METHOD PUBLIC Clone : I_Node
VAR
	pNode : POINTER TO NE_LWORD;
END_VAR
pNode := __NEW(NE_LWORD);
Clone := pNode^;
END_METHOD

METHOD FB_init : BOOL
VAR_INPUT
	bInitRetains : BOOL; // if TRUE, the retain variables are initialized (warm start / cold start)
	bInCopyCode : BOOL;  // if TRUE, the instance afterwards gets moved into the copy code (online change)
END_VAR
AddInput('in1',THIS^.in1);
AddInput('in2',THIS^.in2);
AddOutput('out', THIS^.out);
END_METHOD

METHOD PROTECTED OnExecute
VAR
END_VAR
out.Value := in1.Value <> in2.Value;
END_METHOD

END_FUNCTION_BLOCK

// ---- Comparison/Nodes/NE/NE_REAL.TcPOU
{attribute 'linkalways'} 
{attribute 'no_explicit_call' := 'This FB is a CLASS and must be accessed using methods or properties'}
{attribute 'enable_dynamic_creation'}
FUNCTION_BLOCK FINAL NE_REAL EXTENDS Node
VAR
	in1 : _REAL(0.0);
	in2 : _REAL(0.0);
	out : _BOOL(FALSE);
END_VAR

METHOD PUBLIC Clone : I_Node
VAR
	pNode : POINTER TO NE_REAL;
END_VAR
pNode := __NEW(NE_REAL);
Clone := pNode^;
END_METHOD

METHOD FB_init : BOOL
VAR_INPUT
	bInitRetains : BOOL; // if TRUE, the retain variables are initialized (warm start / cold start)
	bInCopyCode : BOOL;  // if TRUE, the instance afterwards gets moved into the copy code (online change)
END_VAR
AddInput('in1',THIS^.in1);
AddInput('in2',THIS^.in2);
AddOutput('out', THIS^.out);
END_METHOD

METHOD PROTECTED OnExecute
VAR
END_VAR
out.Value := in1.Value <> in2.Value;
END_METHOD

END_FUNCTION_BLOCK

// ---- Comparison/Nodes/NE/NE_SINT.TcPOU
{attribute 'linkalways'} 
{attribute 'no_explicit_call' := 'This FB is a CLASS and must be accessed using methods or properties'}
{attribute 'enable_dynamic_creation'}
FUNCTION_BLOCK FINAL NE_SINT EXTENDS Node
VAR
	in1 : _SINT(0);
	in2 : _SINT(0);
	out : _BOOL(FALSE);
END_VAR

METHOD PUBLIC Clone : I_Node
VAR
	pNode : POINTER TO NE_SINT;
END_VAR
pNode := __NEW(NE_SINT);
Clone := pNode^;
END_METHOD

METHOD FB_init : BOOL
VAR_INPUT
	bInitRetains : BOOL; // if TRUE, the retain variables are initialized (warm start / cold start)
	bInCopyCode : BOOL;  // if TRUE, the instance afterwards gets moved into the copy code (online change)
END_VAR
AddInput('in1',THIS^.in1);
AddInput('in2',THIS^.in2);
AddOutput('out', THIS^.out);
END_METHOD

METHOD PROTECTED OnExecute
VAR
END_VAR
out.Value := in1.Value <> in2.Value;
END_METHOD

END_FUNCTION_BLOCK

// ---- Comparison/Nodes/NE/NE_UDINT.TcPOU
{attribute 'linkalways'} 
{attribute 'no_explicit_call' := 'This FB is a CLASS and must be accessed using methods or properties'}
{attribute 'enable_dynamic_creation'}
FUNCTION_BLOCK FINAL NE_UDINT EXTENDS Node
VAR
	in1 : _UDINT(0);
	in2 : _UDINT(0);
	out : _BOOL(FALSE);
END_VAR

METHOD PUBLIC Clone : I_Node
VAR
	pNode : POINTER TO NE_UDINT;
END_VAR
pNode := __NEW(NE_UDINT);
Clone := pNode^;
END_METHOD

METHOD FB_init : BOOL
VAR_INPUT
	bInitRetains : BOOL; // if TRUE, the retain variables are initialized (warm start / cold start)
	bInCopyCode : BOOL;  // if TRUE, the instance afterwards gets moved into the copy code (online change)
END_VAR
AddInput('in1',THIS^.in1);
AddInput('in2',THIS^.in2);
AddOutput('out', THIS^.out);
END_METHOD

METHOD PROTECTED OnExecute
VAR
END_VAR
out.Value := in1.Value <> in2.Value;
END_METHOD

END_FUNCTION_BLOCK

// ---- Comparison/Nodes/NE/NE_UINT.TcPOU
{attribute 'linkalways'} 
{attribute 'no_explicit_call' := 'This FB is a CLASS and must be accessed using methods or properties'}
{attribute 'enable_dynamic_creation'}
FUNCTION_BLOCK FINAL NE_UINT EXTENDS Node
VAR
	in1 : _UINT(0);
	in2 : _UINT(0);
	out : _BOOL(FALSE);
END_VAR

METHOD PUBLIC Clone : I_Node
VAR
	pNode : POINTER TO NE_UINT;
END_VAR
pNode := __NEW(NE_UINT);
Clone := pNode^;
END_METHOD

METHOD FB_init : BOOL
VAR_INPUT
	bInitRetains : BOOL; // if TRUE, the retain variables are initialized (warm start / cold start)
	bInCopyCode : BOOL;  // if TRUE, the instance afterwards gets moved into the copy code (online change)
END_VAR
AddInput('in1',THIS^.in1);
AddInput('in2',THIS^.in2);
AddOutput('out', THIS^.out);
END_METHOD

METHOD PROTECTED OnExecute
VAR
END_VAR
out.Value := in1.Value <> in2.Value;
END_METHOD

END_FUNCTION_BLOCK

// ---- Comparison/Nodes/NE/NE_ULINT.TcPOU
{attribute 'linkalways'} 
{attribute 'no_explicit_call' := 'This FB is a CLASS and must be accessed using methods or properties'}
{attribute 'enable_dynamic_creation'}
FUNCTION_BLOCK FINAL NE_ULINT EXTENDS Node
VAR
	in1 : _ULINT(0);
	in2 : _ULINT(0);
	out : _BOOL(FALSE);
END_VAR

METHOD PUBLIC Clone : I_Node
VAR
	pNode : POINTER TO NE_ULINT;
END_VAR
pNode := __NEW(NE_ULINT);
Clone := pNode^;
END_METHOD

METHOD FB_init : BOOL
VAR_INPUT
	bInitRetains : BOOL; // if TRUE, the retain variables are initialized (warm start / cold start)
	bInCopyCode : BOOL;  // if TRUE, the instance afterwards gets moved into the copy code (online change)
END_VAR
AddInput('in1',THIS^.in1);
AddInput('in2',THIS^.in2);
AddOutput('out', THIS^.out);
END_METHOD

METHOD PROTECTED OnExecute
VAR
END_VAR
out.Value := in1.Value <> in2.Value;
END_METHOD

END_FUNCTION_BLOCK

// ---- Comparison/Nodes/NE/NE_USINT.TcPOU
{attribute 'linkalways'} 
{attribute 'no_explicit_call' := 'This FB is a CLASS and must be accessed using methods or properties'}
{attribute 'enable_dynamic_creation'}
FUNCTION_BLOCK FINAL NE_USINT EXTENDS Node
VAR
	in1 : _USINT(0);
	in2 : _USINT(0);
	out : _BOOL(FALSE);
END_VAR

METHOD PUBLIC Clone : I_Node
VAR
	pNode : POINTER TO NE_USINT;
END_VAR
pNode := __NEW(NE_USINT);
Clone := pNode^;
END_METHOD

METHOD FB_init : BOOL
VAR_INPUT
	bInitRetains : BOOL; // if TRUE, the retain variables are initialized (warm start / cold start)
	bInCopyCode : BOOL;  // if TRUE, the instance afterwards gets moved into the copy code (online change)
END_VAR
AddInput('in1',THIS^.in1);
AddInput('in2',THIS^.in2);
AddOutput('out', THIS^.out);
END_METHOD

METHOD PROTECTED OnExecute
VAR
END_VAR
out.Value := in1.Value <> in2.Value;
END_METHOD

END_FUNCTION_BLOCK

// ---- Comparison/Nodes/NE/NE_WORD.TcPOU
{attribute 'linkalways'} 
{attribute 'no_explicit_call' := 'This FB is a CLASS and must be accessed using methods or properties'}
{attribute 'enable_dynamic_creation'}
FUNCTION_BLOCK FINAL NE_WORD EXTENDS Node
VAR
	in1 : _WORD(0);
	in2 : _WORD(0);
	out : _BOOL(FALSE);
END_VAR

METHOD PUBLIC Clone : I_Node
VAR
	pNode : POINTER TO NE_WORD;
END_VAR
pNode := __NEW(NE_WORD);
Clone := pNode^;
END_METHOD

METHOD FB_init : BOOL
VAR_INPUT
	bInitRetains : BOOL; // if TRUE, the retain variables are initialized (warm start / cold start)
	bInCopyCode : BOOL;  // if TRUE, the instance afterwards gets moved into the copy code (online change)
END_VAR
AddInput('in1',THIS^.in1);
AddInput('in2',THIS^.in2);
AddOutput('out', THIS^.out);
END_METHOD

METHOD PROTECTED OnExecute
VAR
END_VAR
out.Value := in1.Value <> in2.Value;
END_METHOD

END_FUNCTION_BLOCK

// ---- Core/MathCorePack.TcPOU
{attribute 'linkalways'} 
{attribute 'no_explicit_call' := 'This FB is a CLASS and must be accessed using methods or properties'}
{attribute 'enable_dynamic_creation'}
FUNCTION_BLOCK MathCorePack IMPLEMENTS I_GraphPack
VAR
	ADD_BYTE : ADD_BYTE;
	ADD_DINT : ADD_DINT;
	ADD_DWORD : ADD_DWORD;
	ADD_INT : ADD_INT;
	ADD_LINT : ADD_LINT;
	ADD_LREAL : ADD_LREAL;
	ADD_LWORD : ADD_LWORD;
	ADD_REAL : ADD_REAL;
	ADD_SINT : ADD_SINT;
	ADD_UDINT : ADD_UDINT;
	ADD_UINT : ADD_UINT;
	ADD_ULINT : ADD_ULINT;
	ADD_USINT : ADD_USINT;
	ADD_WORD : ADD_WORD;
	
	SUB_BYTE : SUB_BYTE;
	SUB_DINT : SUB_DINT;
	SUB_DWORD : SUB_DWORD;
	SUB_INT : SUB_INT;
	SUB_LINT : SUB_LINT;
	SUB_LREAL : SUB_LREAL;
	SUB_LWORD : SUB_LWORD;
	SUB_REAL : SUB_REAL;
	SUB_SINT : SUB_SINT;
	SUB_UDINT : SUB_UDINT;
	SUB_UINT : SUB_UINT;
	SUB_ULINT : SUB_ULINT;
	SUB_USINT : SUB_USINT;
	SUB_WORD : SUB_WORD;
	
	MUL_BYTE : MUL_BYTE;
	MUL_DINT : MUL_DINT;
	MUL_DWORD : MUL_DWORD;
	MUL_INT : MUL_INT;
	MUL_LINT : MUL_LINT;
	MUL_LREAL : MUL_LREAL;
	MUL_LWORD : MUL_LWORD;
	MUL_REAL : MUL_REAL;
	MUL_SINT : MUL_SINT;
	MUL_UDINT : MUL_UDINT;
	MUL_UINT : MUL_UINT;
	MUL_ULINT : MUL_ULINT;
	MUL_USINT : MUL_USINT;
	MUL_WORD : MUL_WORD;
	
	DIV_BYTE : DIV_BYTE;
	DIV_DINT : DIV_DINT;
	DIV_DWORD : DIV_DWORD;
	DIV_INT : DIV_INT;
	DIV_LINT : DIV_LINT;
	DIV_LREAL : DIV_LREAL;
	DIV_LWORD : DIV_LWORD;
	DIV_REAL : DIV_REAL;
	DIV_SINT : DIV_SINT;
	DIV_UDINT : DIV_UDINT;
	DIV_UINT : DIV_UINT;
	DIV_ULINT : DIV_ULINT;
	DIV_USINT : DIV_USINT;
	DIV_WORD : DIV_WORD;
	
	MOD_BYTE : MOD_BYTE;
	MOD_DINT : MOD_DINT;
	MOD_DWORD : MOD_DWORD;
	MOD_INT : MOD_INT;
	MOD_LINT : MOD_LINT;
	MOD_LREAL : MOD_LREAL;
	MOD_LWORD : MOD_LWORD;
	MOD_SINT : MOD_SINT;
	MOD_UDINT : MOD_UDINT;
	MOD_UINT : MOD_UINT;
	MOD_ULINT : MOD_ULINT;
	MOD_USINT : MOD_USINT;
	MOD_WORD : MOD_WORD;
	

END_VAR

METHOD Register
VAR_INPUT
	Datatypes : I_Datatypes;
	NodeFactory : I_NodeFactory;
END_VAR
NodeFactory.AddNodeAsPrototype('Math/Core/ADD/ADD_BYTE',ADD_BYTE);
NodeFactory.AddNodeAsPrototype('Math/Core/ADD/ADD_DINT',ADD_DINT);
NodeFactory.AddNodeAsPrototype('Math/Core/ADD/ADD_DWORD',ADD_DWORD);
NodeFactory.AddNodeAsPrototype('Math/Core/ADD/ADD_INT',ADD_INT);
NodeFactory.AddNodeAsPrototype('Math/Core/ADD/ADD_LINT',ADD_LINT);
NodeFactory.AddNodeAsPrototype('Math/Core/ADD/ADD_LREAL',ADD_LREAL);
NodeFactory.AddNodeAsPrototype('Math/Core/ADD/ADD_LWORD',ADD_LWORD);
NodeFactory.AddNodeAsPrototype('Math/Core/ADD/ADD_REAL',ADD_REAL);
NodeFactory.AddNodeAsPrototype('Math/Core/ADD/ADD_SINT',ADD_SINT);
NodeFactory.AddNodeAsPrototype('Math/Core/ADD/ADD_UDINT',ADD_UDINT);
NodeFactory.AddNodeAsPrototype('Math/Core/ADD/ADD_UINT',ADD_UINT);
NodeFactory.AddNodeAsPrototype('Math/Core/ADD/ADD_ULINT',ADD_ULINT);
NodeFactory.AddNodeAsPrototype('Math/Core/ADD/ADD_USINT',ADD_USINT);
NodeFactory.AddNodeAsPrototype('Math/Core/ADD/ADD_WORD',ADD_WORD);

NodeFactory.AddNodeAsPrototype('Math/Core/SUB/SUB_BYTE',SUB_BYTE);
NodeFactory.AddNodeAsPrototype('Math/Core/SUB/SUB_DINT',SUB_DINT);
NodeFactory.AddNodeAsPrototype('Math/Core/SUB/SUB_DWORD',SUB_DWORD);
NodeFactory.AddNodeAsPrototype('Math/Core/SUB/SUB_INT',SUB_INT);
NodeFactory.AddNodeAsPrototype('Math/Core/SUB/SUB_LINT',SUB_LINT);
NodeFactory.AddNodeAsPrototype('Math/Core/SUB/SUB_LREAL',SUB_LREAL);
NodeFactory.AddNodeAsPrototype('Math/Core/SUB/SUB_LWORD',SUB_LWORD);
NodeFactory.AddNodeAsPrototype('Math/Core/SUB/SUB_REAL',SUB_REAL);
NodeFactory.AddNodeAsPrototype('Math/Core/SUB/SUB_SINT',SUB_SINT);
NodeFactory.AddNodeAsPrototype('Math/Core/SUB/SUB_UDINT',SUB_UDINT);
NodeFactory.AddNodeAsPrototype('Math/Core/SUB/SUB_UINT',SUB_UINT);
NodeFactory.AddNodeAsPrototype('Math/Core/SUB/SUB_ULINT',SUB_ULINT);
NodeFactory.AddNodeAsPrototype('Math/Core/SUB/SUB_USINT',SUB_USINT);
NodeFactory.AddNodeAsPrototype('Math/Core/SUB/SUB_WORD',SUB_WORD);

NodeFactory.AddNodeAsPrototype('Math/Core/MUL/MUL_BYTE',MUL_BYTE);
NodeFactory.AddNodeAsPrototype('Math/Core/MUL/MUL_DINT',MUL_DINT);
NodeFactory.AddNodeAsPrototype('Math/Core/MUL/MUL_DWORD',MUL_DWORD);
NodeFactory.AddNodeAsPrototype('Math/Core/MUL/MUL_INT',MUL_INT);
NodeFactory.AddNodeAsPrototype('Math/Core/MUL/MUL_LINT',MUL_LINT);
NodeFactory.AddNodeAsPrototype('Math/Core/MUL/MUL_LREAL',MUL_LREAL);
NodeFactory.AddNodeAsPrototype('Math/Core/MUL/MUL_LWORD',MUL_LWORD);
NodeFactory.AddNodeAsPrototype('Math/Core/MUL/MUL_REAL',MUL_REAL);
NodeFactory.AddNodeAsPrototype('Math/Core/MUL/MUL_SINT',MUL_SINT);
NodeFactory.AddNodeAsPrototype('Math/Core/MUL/MUL_UDINT',MUL_UDINT);
NodeFactory.AddNodeAsPrototype('Math/Core/MUL/MUL_UINT',MUL_UINT);
NodeFactory.AddNodeAsPrototype('Math/Core/MUL/MUL_ULINT',MUL_ULINT);
NodeFactory.AddNodeAsPrototype('Math/Core/MUL/MUL_USINT',MUL_USINT);
NodeFactory.AddNodeAsPrototype('Math/Core/MUL/MUL_WORD',MUL_WORD);

NodeFactory.AddNodeAsPrototype('Math/Core/DIV/DIV_BYTE',DIV_BYTE);
NodeFactory.AddNodeAsPrototype('Math/Core/DIV/DIV_DINT',DIV_DINT);
NodeFactory.AddNodeAsPrototype('Math/Core/DIV/DIV_DWORD',DIV_DWORD);
NodeFactory.AddNodeAsPrototype('Math/Core/DIV/DIV_INT',DIV_INT);
NodeFactory.AddNodeAsPrototype('Math/Core/DIV/DIV_LINT',DIV_LINT);
NodeFactory.AddNodeAsPrototype('Math/Core/DIV/DIV_LREAL',DIV_LREAL);
NodeFactory.AddNodeAsPrototype('Math/Core/DIV/DIV_LWORD',DIV_LWORD);
NodeFactory.AddNodeAsPrototype('Math/Core/DIV/DIV_REAL',DIV_REAL);
NodeFactory.AddNodeAsPrototype('Math/Core/DIV/DIV_SINT',DIV_SINT);
NodeFactory.AddNodeAsPrototype('Math/Core/DIV/DIV_UDINT',DIV_UDINT);
NodeFactory.AddNodeAsPrototype('Math/Core/DIV/DIV_UINT',DIV_UINT);
NodeFactory.AddNodeAsPrototype('Math/Core/DIV/DIV_ULINT',DIV_ULINT);
NodeFactory.AddNodeAsPrototype('Math/Core/DIV/DIV_USINT',DIV_USINT);
NodeFactory.AddNodeAsPrototype('Math/Core/DIV/DIV_WORD',DIV_WORD);

NodeFactory.AddNodeAsPrototype('Math/Core/MOD/MOD_BYTE',MOD_BYTE);
NodeFactory.AddNodeAsPrototype('Math/Core/MOD/MOD_DINT',MOD_DINT);
NodeFactory.AddNodeAsPrototype('Math/Core/MOD/MOD_DWORD',MOD_DWORD);
NodeFactory.AddNodeAsPrototype('Math/Core/MOD/MOD_INT',MOD_INT);
NodeFactory.AddNodeAsPrototype('Math/Core/MOD/MOD_LINT',MOD_LINT);
NodeFactory.AddNodeAsPrototype('Math/Core/MOD/MOD_LREAL',MOD_LREAL);
NodeFactory.AddNodeAsPrototype('Math/Core/MOD/MOD_LWORD',MOD_LWORD);
NodeFactory.AddNodeAsPrototype('Math/Core/MOD/MOD_SINT',MOD_SINT);
NodeFactory.AddNodeAsPrototype('Math/Core/MOD/MOD_UDINT',MOD_UDINT);
NodeFactory.AddNodeAsPrototype('Math/Core/MOD/MOD_UINT',MOD_UINT);
NodeFactory.AddNodeAsPrototype('Math/Core/MOD/MOD_ULINT',MOD_ULINT);
NodeFactory.AddNodeAsPrototype('Math/Core/MOD/MOD_USINT',MOD_USINT);
NodeFactory.AddNodeAsPrototype('Math/Core/MOD/MOD_WORD',MOD_WORD);
END_METHOD

END_FUNCTION_BLOCK

// ---- Core/Nodes/ADD/ADD_BYTE.TcPOU
{attribute 'linkalways'} 
{attribute 'no_explicit_call' := 'This FB is a CLASS and must be accessed using methods or properties'}
{attribute 'enable_dynamic_creation'}
FUNCTION_BLOCK FINAL ADD_BYTE EXTENDS Node
VAR
	in1 : _BYTE(0);
	in2 : _BYTE(0);
	out : _BYTE(0);
END_VAR

METHOD PUBLIC Clone : I_Node
VAR
	pNode : POINTER TO ADD_BYTE;
END_VAR
pNode := __NEW(ADD_BYTE);
Clone := pNode^;
END_METHOD

METHOD FB_init : BOOL
VAR_INPUT
	bInitRetains : BOOL; // if TRUE, the retain variables are initialized (warm start / cold start)
	bInCopyCode : BOOL;  // if TRUE, the instance afterwards gets moved into the copy code (online change)
END_VAR
AddInput('in1',THIS^.in1);
AddInput('in2',THIS^.in2);
AddOutput('out', THIS^.out);
END_METHOD

METHOD PROTECTED OnExecute
VAR
END_VAR
out.Value := in1.Value + in2.Value;
END_METHOD

END_FUNCTION_BLOCK

// ---- Core/Nodes/ADD/ADD_DINT.TcPOU
{attribute 'linkalways'} 
{attribute 'no_explicit_call' := 'This FB is a CLASS and must be accessed using methods or properties'}
{attribute 'enable_dynamic_creation'}
FUNCTION_BLOCK FINAL ADD_DINT EXTENDS Node
VAR
	in1 : _DINT(0);
	in2 : _DINT(0);
	out : _DINT(0);
END_VAR

METHOD PUBLIC Clone : I_Node
VAR
	pNode : POINTER TO ADD_DINT;
END_VAR
pNode := __NEW(ADD_DINT);
Clone := pNode^;
END_METHOD

METHOD FB_init : BOOL
VAR_INPUT
	bInitRetains : BOOL; // if TRUE, the retain variables are initialized (warm start / cold start)
	bInCopyCode : BOOL;  // if TRUE, the instance afterwards gets moved into the copy code (online change)
END_VAR
AddInput('in1',THIS^.in1);
AddInput('in2',THIS^.in2);
AddOutput('out', THIS^.out);
END_METHOD

METHOD PROTECTED OnExecute
VAR
END_VAR
out.Value := in1.Value + in2.Value;
END_METHOD

END_FUNCTION_BLOCK

// ---- Core/Nodes/ADD/ADD_DWORD.TcPOU
{attribute 'linkalways'} 
{attribute 'no_explicit_call' := 'This FB is a CLASS and must be accessed using methods or properties'}
{attribute 'enable_dynamic_creation'}
FUNCTION_BLOCK FINAL ADD_DWORD EXTENDS Node
VAR
	in1 : _DWORD(0);
	in2 : _DWORD(0);
	out : _DWORD(0);
END_VAR

METHOD PUBLIC Clone : I_Node
VAR
	pNode : POINTER TO ADD_DWORD;
END_VAR
pNode := __NEW(ADD_DWORD);
Clone := pNode^;
END_METHOD

METHOD FB_init : BOOL
VAR_INPUT
	bInitRetains : BOOL; // if TRUE, the retain variables are initialized (warm start / cold start)
	bInCopyCode : BOOL;  // if TRUE, the instance afterwards gets moved into the copy code (online change)
END_VAR
AddInput('in1',THIS^.in1);
AddInput('in2',THIS^.in2);
AddOutput('out', THIS^.out);
END_METHOD

METHOD PROTECTED OnExecute
VAR
END_VAR
out.Value := in1.Value + in2.Value;
END_METHOD

END_FUNCTION_BLOCK

// ---- Core/Nodes/ADD/ADD_INT.TcPOU
{attribute 'linkalways'} 
{attribute 'no_explicit_call' := 'This FB is a CLASS and must be accessed using methods or properties'}
{attribute 'enable_dynamic_creation'}
FUNCTION_BLOCK FINAL ADD_INT EXTENDS Node
VAR
	in1 : _INT(0);
	in2 : _INT(0);
	out : _INT(0);
END_VAR

METHOD PUBLIC Clone : I_Node
VAR
	pNode : POINTER TO ADD_INT;
END_VAR
pNode := __NEW(ADD_INT);
Clone := pNode^;
END_METHOD

METHOD FB_init : BOOL
VAR_INPUT
	bInitRetains : BOOL; // if TRUE, the retain variables are initialized (warm start / cold start)
	bInCopyCode : BOOL;  // if TRUE, the instance afterwards gets moved into the copy code (online change)
END_VAR
AddInput('in1',THIS^.in1);
AddInput('in2',THIS^.in2);
AddOutput('out', THIS^.out);
END_METHOD

METHOD PROTECTED OnExecute
VAR
END_VAR
out.Value := in1.Value + in2.Value;
END_METHOD

END_FUNCTION_BLOCK

// ---- Core/Nodes/ADD/ADD_LINT.TcPOU
{attribute 'linkalways'} 
{attribute 'no_explicit_call' := 'This FB is a CLASS and must be accessed using methods or properties'}
{attribute 'enable_dynamic_creation'}
FUNCTION_BLOCK FINAL ADD_LINT EXTENDS Node
VAR
	in1 : _LINT(0);
	in2 : _LINT(0);
	out : _LINT(0);
END_VAR

METHOD PUBLIC Clone : I_Node
VAR
	pNode : POINTER TO ADD_LINT;
END_VAR
pNode := __NEW(ADD_LINT);
Clone := pNode^;
END_METHOD

METHOD FB_init : BOOL
VAR_INPUT
	bInitRetains : BOOL; // if TRUE, the retain variables are initialized (warm start / cold start)
	bInCopyCode : BOOL;  // if TRUE, the instance afterwards gets moved into the copy code (online change)
END_VAR
AddInput('in1',THIS^.in1);
AddInput('in2',THIS^.in2);
AddOutput('out', THIS^.out);
END_METHOD

METHOD PROTECTED OnExecute
VAR
END_VAR
out.Value := in1.Value + in2.Value;
END_METHOD

END_FUNCTION_BLOCK

// ---- Core/Nodes/ADD/ADD_LREAL.TcPOU
{attribute 'linkalways'} 
{attribute 'no_explicit_call' := 'This FB is a CLASS and must be accessed using methods or properties'}
{attribute 'enable_dynamic_creation'}
FUNCTION_BLOCK FINAL ADD_LREAL EXTENDS Node
VAR
	in1 : _LREAL(0.0);
	in2 : _LREAL(0.0);
	out : _LREAL(0.0);
END_VAR

METHOD PUBLIC Clone : I_Node
VAR
	pNode : POINTER TO ADD_LREAL;
END_VAR
pNode := __NEW(ADD_LREAL);
Clone := pNode^;
END_METHOD

METHOD FB_init : BOOL
VAR_INPUT
	bInitRetains : BOOL; // if TRUE, the retain variables are initialized (warm start / cold start)
	bInCopyCode : BOOL;  // if TRUE, the instance afterwards gets moved into the copy code (online change)
END_VAR
AddInput('in1',THIS^.in1);
AddInput('in2',THIS^.in2);
AddOutput('out', THIS^.out);
END_METHOD

METHOD PROTECTED OnExecute
VAR
END_VAR
out.Value := in1.Value + in2.Value;
END_METHOD

END_FUNCTION_BLOCK

// ---- Core/Nodes/ADD/ADD_LWORD.TcPOU
{attribute 'linkalways'} 
{attribute 'no_explicit_call' := 'This FB is a CLASS and must be accessed using methods or properties'}
{attribute 'enable_dynamic_creation'}
FUNCTION_BLOCK FINAL ADD_LWORD EXTENDS Node
VAR
	in1 : _LWORD(0);
	in2 : _LWORD(0);
	out : _LWORD(0);
END_VAR

METHOD PUBLIC Clone : I_Node
VAR
	pNode : POINTER TO ADD_LWORD;
END_VAR
pNode := __NEW(ADD_LWORD);
Clone := pNode^;
END_METHOD

METHOD FB_init : BOOL
VAR_INPUT
	bInitRetains : BOOL; // if TRUE, the retain variables are initialized (warm start / cold start)
	bInCopyCode : BOOL;  // if TRUE, the instance afterwards gets moved into the copy code (online change)
END_VAR
AddInput('in1',THIS^.in1);
AddInput('in2',THIS^.in2);
AddOutput('out', THIS^.out);
END_METHOD

METHOD PROTECTED OnExecute
VAR
END_VAR
out.Value := in1.Value + in2.Value;
END_METHOD

END_FUNCTION_BLOCK

// ---- Core/Nodes/ADD/ADD_REAL.TcPOU
{attribute 'linkalways'} 
{attribute 'no_explicit_call' := 'This FB is a CLASS and must be accessed using methods or properties'}
{attribute 'enable_dynamic_creation'}
FUNCTION_BLOCK FINAL ADD_REAL EXTENDS Node
VAR
	in1 : _REAL(0.0);
	in2 : _REAL(0.0);
	out : _REAL(0.0);
END_VAR

METHOD PUBLIC Clone : I_Node
VAR
	pNode : POINTER TO ADD_REAL;
END_VAR
pNode := __NEW(ADD_REAL);
Clone := pNode^;
END_METHOD

METHOD FB_init : BOOL
VAR_INPUT
	bInitRetains : BOOL; // if TRUE, the retain variables are initialized (warm start / cold start)
	bInCopyCode : BOOL;  // if TRUE, the instance afterwards gets moved into the copy code (online change)
END_VAR
AddInput('in1',THIS^.in1);
AddInput('in2',THIS^.in2);
AddOutput('out', THIS^.out);
END_METHOD

METHOD PROTECTED OnExecute
VAR
END_VAR
out.Value := in1.Value + in2.Value;
END_METHOD

END_FUNCTION_BLOCK

// ---- Core/Nodes/ADD/ADD_SINT.TcPOU
{attribute 'linkalways'} 
{attribute 'no_explicit_call' := 'This FB is a CLASS and must be accessed using methods or properties'}
{attribute 'enable_dynamic_creation'}
FUNCTION_BLOCK FINAL ADD_SINT EXTENDS Node
VAR
	in1 : _SINT(0);
	in2 : _SINT(0);
	out : _SINT(0);
END_VAR

METHOD PUBLIC Clone : I_Node
VAR
	pNode : POINTER TO ADD_SINT;
END_VAR
pNode := __NEW(ADD_SINT);
Clone := pNode^;
END_METHOD

METHOD FB_init : BOOL
VAR_INPUT
	bInitRetains : BOOL; // if TRUE, the retain variables are initialized (warm start / cold start)
	bInCopyCode : BOOL;  // if TRUE, the instance afterwards gets moved into the copy code (online change)
END_VAR
AddInput('in1',THIS^.in1);
AddInput('in2',THIS^.in2);
AddOutput('out', THIS^.out);
END_METHOD

METHOD PROTECTED OnExecute
VAR
END_VAR
out.Value := in1.Value + in2.Value;
END_METHOD

END_FUNCTION_BLOCK

// ---- Core/Nodes/ADD/ADD_UDINT.TcPOU
{attribute 'linkalways'} 
{attribute 'no_explicit_call' := 'This FB is a CLASS and must be accessed using methods or properties'}
{attribute 'enable_dynamic_creation'}
FUNCTION_BLOCK FINAL ADD_UDINT EXTENDS Node
VAR
	in1 : _UDINT(0);
	in2 : _UDINT(0);
	out : _UDINT(0);
END_VAR

METHOD PUBLIC Clone : I_Node
VAR
	pNode : POINTER TO ADD_UDINT;
END_VAR
pNode := __NEW(ADD_UDINT);
Clone := pNode^;
END_METHOD

METHOD FB_init : BOOL
VAR_INPUT
	bInitRetains : BOOL; // if TRUE, the retain variables are initialized (warm start / cold start)
	bInCopyCode : BOOL;  // if TRUE, the instance afterwards gets moved into the copy code (online change)
END_VAR
AddInput('in1',THIS^.in1);
AddInput('in2',THIS^.in2);
AddOutput('out', THIS^.out);
END_METHOD

METHOD PROTECTED OnExecute
VAR
END_VAR
out.Value := in1.Value + in2.Value;
END_METHOD

END_FUNCTION_BLOCK

// ---- Core/Nodes/ADD/ADD_UINT.TcPOU
{attribute 'linkalways'} 
{attribute 'no_explicit_call' := 'This FB is a CLASS and must be accessed using methods or properties'}
{attribute 'enable_dynamic_creation'}
FUNCTION_BLOCK FINAL ADD_UINT EXTENDS Node
VAR
	in1 : _UINT(0);
	in2 : _UINT(0);
	out : _UINT(0);
END_VAR

METHOD PUBLIC Clone : I_Node
VAR
	pNode : POINTER TO ADD_UINT;
END_VAR
pNode := __NEW(ADD_UINT);
Clone := pNode^;
END_METHOD

METHOD FB_init : BOOL
VAR_INPUT
	bInitRetains : BOOL; // if TRUE, the retain variables are initialized (warm start / cold start)
	bInCopyCode : BOOL;  // if TRUE, the instance afterwards gets moved into the copy code (online change)
END_VAR
AddInput('in1',THIS^.in1);
AddInput('in2',THIS^.in2);
AddOutput('out', THIS^.out);
END_METHOD

METHOD PROTECTED OnExecute
VAR
END_VAR
out.Value := in1.Value + in2.Value;
END_METHOD

END_FUNCTION_BLOCK

// ---- Core/Nodes/ADD/ADD_ULINT.TcPOU
{attribute 'linkalways'} 
{attribute 'no_explicit_call' := 'This FB is a CLASS and must be accessed using methods or properties'}
{attribute 'enable_dynamic_creation'}
FUNCTION_BLOCK FINAL ADD_ULINT EXTENDS Node
VAR
	in1 : _ULINT(0);
	in2 : _ULINT(0);
	out : _ULINT(0);
END_VAR

METHOD PUBLIC Clone : I_Node
VAR
	pNode : POINTER TO ADD_ULINT;
END_VAR
pNode := __NEW(ADD_ULINT);
Clone := pNode^;
END_METHOD

METHOD FB_init : BOOL
VAR_INPUT
	bInitRetains : BOOL; // if TRUE, the retain variables are initialized (warm start / cold start)
	bInCopyCode : BOOL;  // if TRUE, the instance afterwards gets moved into the copy code (online change)
END_VAR
AddInput('in1',THIS^.in1);
AddInput('in2',THIS^.in2);
AddOutput('out', THIS^.out);
END_METHOD

METHOD PROTECTED OnExecute
VAR
END_VAR
out.Value := in1.Value + in2.Value;
END_METHOD

END_FUNCTION_BLOCK

// ---- Core/Nodes/ADD/ADD_USINT.TcPOU
{attribute 'linkalways'} 
{attribute 'no_explicit_call' := 'This FB is a CLASS and must be accessed using methods or properties'}
{attribute 'enable_dynamic_creation'}
FUNCTION_BLOCK FINAL ADD_USINT EXTENDS Node
VAR
	in1 : _USINT(0);
	in2 : _USINT(0);
	out : _USINT(0);
END_VAR

METHOD PUBLIC Clone : I_Node
VAR
	pNode : POINTER TO ADD_USINT;
END_VAR
pNode := __NEW(ADD_USINT);
Clone := pNode^;
END_METHOD

METHOD FB_init : BOOL
VAR_INPUT
	bInitRetains : BOOL; // if TRUE, the retain variables are initialized (warm start / cold start)
	bInCopyCode : BOOL;  // if TRUE, the instance afterwards gets moved into the copy code (online change)
END_VAR
AddInput('in1',THIS^.in1);
AddInput('in2',THIS^.in2);
AddOutput('out', THIS^.out);
END_METHOD

METHOD PROTECTED OnExecute
VAR
END_VAR
out.Value := in1.Value + in2.Value;
END_METHOD

END_FUNCTION_BLOCK

// ---- Core/Nodes/ADD/ADD_WORD.TcPOU
{attribute 'linkalways'} 
{attribute 'no_explicit_call' := 'This FB is a CLASS and must be accessed using methods or properties'}
{attribute 'enable_dynamic_creation'}
FUNCTION_BLOCK FINAL ADD_WORD EXTENDS Node
VAR
	in1 : _WORD(0);
	in2 : _WORD(0);
	out : _WORD(0);
END_VAR

METHOD PUBLIC Clone : I_Node
VAR
	pNode : POINTER TO ADD_WORD;
END_VAR
pNode := __NEW(ADD_WORD);
Clone := pNode^;
END_METHOD

METHOD FB_init : BOOL
VAR_INPUT
	bInitRetains : BOOL; // if TRUE, the retain variables are initialized (warm start / cold start)
	bInCopyCode : BOOL;  // if TRUE, the instance afterwards gets moved into the copy code (online change)
END_VAR
AddInput('in1',THIS^.in1);
AddInput('in2',THIS^.in2);
AddOutput('out', THIS^.out);
END_METHOD

METHOD PROTECTED OnExecute
VAR
END_VAR
out.Value := in1.Value + in2.Value;
END_METHOD

END_FUNCTION_BLOCK

// ---- Core/Nodes/SUB/SUB_BYTE.TcPOU
{attribute 'linkalways'} 
{attribute 'no_explicit_call' := 'This FB is a CLASS and must be accessed using methods or properties'}
{attribute 'enable_dynamic_creation'}
FUNCTION_BLOCK FINAL SUB_BYTE EXTENDS Node
VAR
	in1 : _BYTE(0);
	in2 : _BYTE(0);
	out : _BYTE(0);
END_VAR

METHOD PUBLIC Clone : I_Node
VAR
	pNode : POINTER TO SUB_BYTE;
END_VAR
pNode := __NEW(SUB_BYTE);
Clone := pNode^;
END_METHOD

METHOD FB_init : BOOL
VAR_INPUT
	bInitRetains : BOOL; // if TRUE, the retain variables are initialized (warm start / cold start)
	bInCopyCode : BOOL;  // if TRUE, the instance afterwards gets moved into the copy code (online change)
END_VAR
AddInput('in1',THIS^.in1);
AddInput('in2',THIS^.in2);
AddOutput('out', THIS^.out);
END_METHOD

METHOD PROTECTED OnExecute
VAR
END_VAR
out.Value := in1.Value - in2.Value;
END_METHOD

END_FUNCTION_BLOCK

// ---- Core/Nodes/SUB/SUB_DINT.TcPOU
{attribute 'linkalways'} 
{attribute 'no_explicit_call' := 'This FB is a CLASS and must be accessed using methods or properties'}
{attribute 'enable_dynamic_creation'}
FUNCTION_BLOCK FINAL SUB_DINT EXTENDS Node
VAR
	in1 : _DINT(0);
	in2 : _DINT(0);
	out : _DINT(0);
END_VAR

METHOD PUBLIC Clone : I_Node
VAR
	pNode : POINTER TO SUB_DINT;
END_VAR
pNode := __NEW(SUB_DINT);
Clone := pNode^;
END_METHOD

METHOD FB_init : BOOL
VAR_INPUT
	bInitRetains : BOOL; // if TRUE, the retain variables are initialized (warm start / cold start)
	bInCopyCode : BOOL;  // if TRUE, the instance afterwards gets moved into the copy code (online change)
END_VAR
AddInput('in1',THIS^.in1);
AddInput('in2',THIS^.in2);
AddOutput('out', THIS^.out);
END_METHOD

METHOD PROTECTED OnExecute
VAR
END_VAR
out.Value := in1.Value - in2.Value;
END_METHOD

END_FUNCTION_BLOCK

// ---- Core/Nodes/SUB/SUB_DWORD.TcPOU
{attribute 'linkalways'} 
{attribute 'no_explicit_call' := 'This FB is a CLASS and must be accessed using methods or properties'}
{attribute 'enable_dynamic_creation'}
FUNCTION_BLOCK FINAL SUB_DWORD EXTENDS Node
VAR
	in1 : _DWORD(0);
	in2 : _DWORD(0);
	out : _DWORD(0);
END_VAR

METHOD PUBLIC Clone : I_Node
VAR
	pNode : POINTER TO SUB_DWORD;
END_VAR
pNode := __NEW(SUB_DWORD);
Clone := pNode^;
END_METHOD

METHOD FB_init : BOOL
VAR_INPUT
	bInitRetains : BOOL; // if TRUE, the retain variables are initialized (warm start / cold start)
	bInCopyCode : BOOL;  // if TRUE, the instance afterwards gets moved into the copy code (online change)
END_VAR
AddInput('in1',THIS^.in1);
AddInput('in2',THIS^.in2);
AddOutput('out', THIS^.out);
END_METHOD

METHOD PROTECTED OnExecute
VAR
END_VAR
out.Value := in1.Value - in2.Value;
END_METHOD

END_FUNCTION_BLOCK

// ---- Core/Nodes/SUB/SUB_INT.TcPOU
{attribute 'linkalways'} 
{attribute 'no_explicit_call' := 'This FB is a CLASS and must be accessed using methods or properties'}
{attribute 'enable_dynamic_creation'}
FUNCTION_BLOCK FINAL SUB_INT EXTENDS Node
VAR
	in1 : _INT(0);
	in2 : _INT(0);
	out : _INT(0);
END_VAR

METHOD PUBLIC Clone : I_Node
VAR
	pNode : POINTER TO SUB_INT;
END_VAR
pNode := __NEW(SUB_INT);
Clone := pNode^;
END_METHOD

METHOD FB_init : BOOL
VAR_INPUT
	bInitRetains : BOOL; // if TRUE, the retain variables are initialized (warm start / cold start)
	bInCopyCode : BOOL;  // if TRUE, the instance afterwards gets moved into the copy code (online change)
END_VAR
AddInput('in1',THIS^.in1);
AddInput('in2',THIS^.in2);
AddOutput('out', THIS^.out);
END_METHOD

METHOD PROTECTED OnExecute
VAR
END_VAR
out.Value := in1.Value - in2.Value;
END_METHOD

END_FUNCTION_BLOCK

// ---- Core/Nodes/SUB/SUB_LINT.TcPOU
{attribute 'linkalways'} 
{attribute 'no_explicit_call' := 'This FB is a CLASS and must be accessed using methods or properties'}
{attribute 'enable_dynamic_creation'}
FUNCTION_BLOCK FINAL SUB_LINT EXTENDS Node
VAR
	in1 : _LINT(0);
	in2 : _LINT(0);
	out : _LINT(0);
END_VAR

METHOD PUBLIC Clone : I_Node
VAR
	pNode : POINTER TO SUB_LINT;
END_VAR
pNode := __NEW(SUB_LINT);
Clone := pNode^;
END_METHOD

METHOD FB_init : BOOL
VAR_INPUT
	bInitRetains : BOOL; // if TRUE, the retain variables are initialized (warm start / cold start)
	bInCopyCode : BOOL;  // if TRUE, the instance afterwards gets moved into the copy code (online change)
END_VAR
AddInput('in1',THIS^.in1);
AddInput('in2',THIS^.in2);
AddOutput('out', THIS^.out);
END_METHOD

METHOD PROTECTED OnExecute
VAR
END_VAR
out.Value := in1.Value - in2.Value;
END_METHOD

END_FUNCTION_BLOCK

// ---- Core/Nodes/SUB/SUB_LREAL.TcPOU
{attribute 'linkalways'} 
{attribute 'no_explicit_call' := 'This FB is a CLASS and must be accessed using methods or properties'}
{attribute 'enable_dynamic_creation'}
FUNCTION_BLOCK FINAL SUB_LREAL EXTENDS Node
VAR
	in1 : _LREAL(0.0);
	in2 : _LREAL(0.0);
	out : _LREAL(0.0);
END_VAR

METHOD PUBLIC Clone : I_Node
VAR
	pNode : POINTER TO SUB_LREAL;
END_VAR
pNode := __NEW(SUB_LREAL);
Clone := pNode^;
END_METHOD

METHOD FB_init : BOOL
VAR_INPUT
	bInitRetains : BOOL; // if TRUE, the retain variables are initialized (warm start / cold start)
	bInCopyCode : BOOL;  // if TRUE, the instance afterwards gets moved into the copy code (online change)
END_VAR
AddInput('in1',THIS^.in1);
AddInput('in2',THIS^.in2);
AddOutput('out', THIS^.out);
END_METHOD

METHOD PROTECTED OnExecute
VAR
END_VAR
out.Value := in1.Value - in2.Value;
END_METHOD

END_FUNCTION_BLOCK

// ---- Core/Nodes/SUB/SUB_LWORD.TcPOU
{attribute 'linkalways'} 
{attribute 'no_explicit_call' := 'This FB is a CLASS and must be accessed using methods or properties'}
{attribute 'enable_dynamic_creation'}
FUNCTION_BLOCK FINAL SUB_LWORD EXTENDS Node
VAR
	in1 : _LWORD(0);
	in2 : _LWORD(0);
	out : _LWORD(0);
END_VAR

METHOD PUBLIC Clone : I_Node
VAR
	pNode : POINTER TO SUB_LWORD;
END_VAR
pNode := __NEW(SUB_LWORD);
Clone := pNode^;
END_METHOD

METHOD FB_init : BOOL
VAR_INPUT
	bInitRetains : BOOL; // if TRUE, the retain variables are initialized (warm start / cold start)
	bInCopyCode : BOOL;  // if TRUE, the instance afterwards gets moved into the copy code (online change)
END_VAR
AddInput('in1',THIS^.in1);
AddInput('in2',THIS^.in2);
AddOutput('out', THIS^.out);
END_METHOD

METHOD PROTECTED OnExecute
VAR
END_VAR
out.Value := in1.Value - in2.Value;
END_METHOD

END_FUNCTION_BLOCK

// ---- Core/Nodes/SUB/SUB_REAL.TcPOU
{attribute 'linkalways'} 
{attribute 'no_explicit_call' := 'This FB is a CLASS and must be accessed using methods or properties'}
{attribute 'enable_dynamic_creation'}
FUNCTION_BLOCK FINAL SUB_REAL EXTENDS Node
VAR
	in1 : _REAL(0.0);
	in2 : _REAL(0.0);
	out : _REAL(0.0);
END_VAR

METHOD PUBLIC Clone : I_Node
VAR
	pNode : POINTER TO SUB_REAL;
END_VAR
pNode := __NEW(SUB_REAL);
Clone := pNode^;
END_METHOD

METHOD FB_init : BOOL
VAR_INPUT
	bInitRetains : BOOL; // if TRUE, the retain variables are initialized (warm start / cold start)
	bInCopyCode : BOOL;  // if TRUE, the instance afterwards gets moved into the copy code (online change)
END_VAR
AddInput('in1',THIS^.in1);
AddInput('in2',THIS^.in2);
AddOutput('out', THIS^.out);
END_METHOD

METHOD PROTECTED OnExecute
VAR
END_VAR
out.Value := in1.Value - in2.Value;
END_METHOD

END_FUNCTION_BLOCK

// ---- Core/Nodes/SUB/SUB_SINT.TcPOU
{attribute 'linkalways'} 
{attribute 'no_explicit_call' := 'This FB is a CLASS and must be accessed using methods or properties'}
{attribute 'enable_dynamic_creation'}
FUNCTION_BLOCK FINAL SUB_SINT EXTENDS Node
VAR
	in1 : _SINT(0);
	in2 : _SINT(0);
	out : _SINT(0);
END_VAR

METHOD PUBLIC Clone : I_Node
VAR
	pNode : POINTER TO SUB_SINT;
END_VAR
pNode := __NEW(SUB_SINT);
Clone := pNode^;
END_METHOD

METHOD FB_init : BOOL
VAR_INPUT
	bInitRetains : BOOL; // if TRUE, the retain variables are initialized (warm start / cold start)
	bInCopyCode : BOOL;  // if TRUE, the instance afterwards gets moved into the copy code (online change)
END_VAR
AddInput('in1',THIS^.in1);
AddInput('in2',THIS^.in2);
AddOutput('out', THIS^.out);
END_METHOD

METHOD PROTECTED OnExecute
VAR
END_VAR
out.Value := in1.Value - in2.Value;
END_METHOD

END_FUNCTION_BLOCK

// ---- Core/Nodes/SUB/SUB_UDINT.TcPOU
{attribute 'linkalways'} 
{attribute 'no_explicit_call' := 'This FB is a CLASS and must be accessed using methods or properties'}
{attribute 'enable_dynamic_creation'}
FUNCTION_BLOCK FINAL SUB_UDINT EXTENDS Node
VAR
	in1 : _UDINT(0);
	in2 : _UDINT(0);
	out : _UDINT(0);
END_VAR

METHOD PUBLIC Clone : I_Node
VAR
	pNode : POINTER TO SUB_UDINT;
END_VAR
pNode := __NEW(SUB_UDINT);
Clone := pNode^;
END_METHOD

METHOD FB_init : BOOL
VAR_INPUT
	bInitRetains : BOOL; // if TRUE, the retain variables are initialized (warm start / cold start)
	bInCopyCode : BOOL;  // if TRUE, the instance afterwards gets moved into the copy code (online change)
END_VAR
AddInput('in1',THIS^.in1);
AddInput('in2',THIS^.in2);
AddOutput('out', THIS^.out);
END_METHOD

METHOD PROTECTED OnExecute
VAR
END_VAR
out.Value := in1.Value - in2.Value;
END_METHOD

END_FUNCTION_BLOCK

// ---- Core/Nodes/SUB/SUB_UINT.TcPOU
{attribute 'linkalways'} 
{attribute 'no_explicit_call' := 'This FB is a CLASS and must be accessed using methods or properties'}
{attribute 'enable_dynamic_creation'}
FUNCTION_BLOCK FINAL SUB_UINT EXTENDS Node
VAR
	in1 : _UINT(0);
	in2 : _UINT(0);
	out : _UINT(0);
END_VAR

METHOD PUBLIC Clone : I_Node
VAR
	pNode : POINTER TO SUB_UINT;
END_VAR
pNode := __NEW(SUB_UINT);
Clone := pNode^;
END_METHOD

METHOD FB_init : BOOL
VAR_INPUT
	bInitRetains : BOOL; // if TRUE, the retain variables are initialized (warm start / cold start)
	bInCopyCode : BOOL;  // if TRUE, the instance afterwards gets moved into the copy code (online change)
END_VAR
AddInput('in1',THIS^.in1);
AddInput('in2',THIS^.in2);
AddOutput('out', THIS^.out);
END_METHOD

METHOD PROTECTED OnExecute
VAR
END_VAR
out.Value := in1.Value - in2.Value;
END_METHOD

END_FUNCTION_BLOCK

// ---- Core/Nodes/SUB/SUB_ULINT.TcPOU
{attribute 'linkalways'} 
{attribute 'no_explicit_call' := 'This FB is a CLASS and must be accessed using methods or properties'}
{attribute 'enable_dynamic_creation'}
FUNCTION_BLOCK FINAL SUB_ULINT EXTENDS Node
VAR
	in1 : _ULINT(0);
	in2 : _ULINT(0);
	out : _ULINT(0);
END_VAR

METHOD PUBLIC Clone : I_Node
VAR
	pNode : POINTER TO SUB_ULINT;
END_VAR
pNode := __NEW(SUB_ULINT);
Clone := pNode^;
END_METHOD

METHOD FB_init : BOOL
VAR_INPUT
	bInitRetains : BOOL; // if TRUE, the retain variables are initialized (warm start / cold start)
	bInCopyCode : BOOL;  // if TRUE, the instance afterwards gets moved into the copy code (online change)
END_VAR
AddInput('in1',THIS^.in1);
AddInput('in2',THIS^.in2);
AddOutput('out', THIS^.out);
END_METHOD

METHOD PROTECTED OnExecute
VAR
END_VAR
out.Value := in1.Value - in2.Value;
END_METHOD

END_FUNCTION_BLOCK

// ---- Core/Nodes/SUB/SUB_USINT.TcPOU
{attribute 'linkalways'} 
{attribute 'no_explicit_call' := 'This FB is a CLASS and must be accessed using methods or properties'}
{attribute 'enable_dynamic_creation'}
FUNCTION_BLOCK FINAL SUB_USINT EXTENDS Node
VAR
	in1 : _USINT(0);
	in2 : _USINT(0);
	out : _USINT(0);
END_VAR

METHOD PUBLIC Clone : I_Node
VAR
	pNode : POINTER TO SUB_USINT;
END_VAR
pNode := __NEW(SUB_USINT);
Clone := pNode^;
END_METHOD

METHOD FB_init : BOOL
VAR_INPUT
	bInitRetains : BOOL; // if TRUE, the retain variables are initialized (warm start / cold start)
	bInCopyCode : BOOL;  // if TRUE, the instance afterwards gets moved into the copy code (online change)
END_VAR
AddInput('in1',THIS^.in1);
AddInput('in2',THIS^.in2);
AddOutput('out', THIS^.out);
END_METHOD

METHOD PROTECTED OnExecute
VAR
END_VAR
out.Value := in1.Value - in2.Value;
END_METHOD

END_FUNCTION_BLOCK

// ---- Core/Nodes/SUB/SUB_WORD.TcPOU
{attribute 'linkalways'} 
{attribute 'no_explicit_call' := 'This FB is a CLASS and must be accessed using methods or properties'}
{attribute 'enable_dynamic_creation'}
FUNCTION_BLOCK FINAL SUB_WORD EXTENDS Node
VAR
	in1 : _WORD(0);
	in2 : _WORD(0);
	out : _WORD(0);
END_VAR

METHOD PUBLIC Clone : I_Node
VAR
	pNode : POINTER TO SUB_WORD;
END_VAR
pNode := __NEW(SUB_WORD);
Clone := pNode^;
END_METHOD

METHOD FB_init : BOOL
VAR_INPUT
	bInitRetains : BOOL; // if TRUE, the retain variables are initialized (warm start / cold start)
	bInCopyCode : BOOL;  // if TRUE, the instance afterwards gets moved into the copy code (online change)
END_VAR
AddInput('in1',THIS^.in1);
AddInput('in2',THIS^.in2);
AddOutput('out', THIS^.out);
END_METHOD

METHOD PROTECTED OnExecute
VAR
END_VAR
out.Value := in1.Value - in2.Value;
END_METHOD

END_FUNCTION_BLOCK

// ---- Core/Nodes/MUL/MUL_BYTE.TcPOU
{attribute 'linkalways'} 
{attribute 'no_explicit_call' := 'This FB is a CLASS and must be accessed using methods or properties'}
{attribute 'enable_dynamic_creation'}
FUNCTION_BLOCK FINAL MUL_BYTE EXTENDS Node
VAR
	in1 : _BYTE(0);
	in2 : _BYTE(0);
	out : _BYTE(0);
END_VAR

METHOD PUBLIC Clone : I_Node
VAR
	pNode : POINTER TO MUL_BYTE;
END_VAR
pNode := __NEW(MUL_BYTE);
Clone := pNode^;
END_METHOD

METHOD FB_init : BOOL
VAR_INPUT
	bInitRetains : BOOL; // if TRUE, the retain variables are initialized (warm start / cold start)
	bInCopyCode : BOOL;  // if TRUE, the instance afterwards gets moved into the copy code (online change)
END_VAR
AddInput('in1',THIS^.in1);
AddInput('in2',THIS^.in2);
AddOutput('out', THIS^.out);
END_METHOD

METHOD PROTECTED OnExecute
VAR
END_VAR
out.Value := in1.Value * in2.Value;
END_METHOD

END_FUNCTION_BLOCK

// ---- Core/Nodes/MUL/MUL_DINT.TcPOU
{attribute 'linkalways'} 
{attribute 'no_explicit_call' := 'This FB is a CLASS and must be accessed using methods or properties'}
{attribute 'enable_dynamic_creation'}
FUNCTION_BLOCK FINAL MUL_DINT EXTENDS Node
VAR
	in1 : _DINT(0);
	in2 : _DINT(0);
	out : _DINT(0);
END_VAR

METHOD PUBLIC Clone : I_Node
VAR
	pNode : POINTER TO MUL_DINT;
END_VAR
pNode := __NEW(MUL_DINT);
Clone := pNode^;
END_METHOD

METHOD FB_init : BOOL
VAR_INPUT
	bInitRetains : BOOL; // if TRUE, the retain variables are initialized (warm start / cold start)
	bInCopyCode : BOOL;  // if TRUE, the instance afterwards gets moved into the copy code (online change)
END_VAR
AddInput('in1',THIS^.in1);
AddInput('in2',THIS^.in2);
AddOutput('out', THIS^.out);
END_METHOD

METHOD PROTECTED OnExecute
VAR
END_VAR
out.Value := in1.Value * in2.Value;
END_METHOD

END_FUNCTION_BLOCK

// ---- Core/Nodes/MUL/MUL_DWORD.TcPOU
{attribute 'linkalways'} 
{attribute 'no_explicit_call' := 'This FB is a CLASS and must be accessed using methods or properties'}
{attribute 'enable_dynamic_creation'}
FUNCTION_BLOCK FINAL MUL_DWORD EXTENDS Node
VAR
	in1 : _DWORD(0);
	in2 : _DWORD(0);
	out : _DWORD(0);
END_VAR

METHOD PUBLIC Clone : I_Node
VAR
	pNode : POINTER TO MUL_DWORD;
END_VAR
pNode := __NEW(MUL_DWORD);
Clone := pNode^;
END_METHOD

METHOD FB_init : BOOL
VAR_INPUT
	bInitRetains : BOOL; // if TRUE, the retain variables are initialized (warm start / cold start)
	bInCopyCode : BOOL;  // if TRUE, the instance afterwards gets moved into the copy code (online change)
END_VAR
AddInput('in1',THIS^.in1);
AddInput('in2',THIS^.in2);
AddOutput('out', THIS^.out);
END_METHOD

METHOD PROTECTED OnExecute
VAR
END_VAR
out.Value := in1.Value * in2.Value;
END_METHOD

END_FUNCTION_BLOCK

// ---- Core/Nodes/MUL/MUL_INT.TcPOU
{attribute 'linkalways'} 
{attribute 'no_explicit_call' := 'This FB is a CLASS and must be accessed using methods or properties'}
{attribute 'enable_dynamic_creation'}
FUNCTION_BLOCK FINAL MUL_INT EXTENDS Node
VAR
	in1 : _INT(0);
	in2 : _INT(0);
	out : _INT(0);
END_VAR

METHOD PUBLIC Clone : I_Node
VAR
	pNode : POINTER TO MUL_INT;
END_VAR
pNode := __NEW(MUL_INT);
Clone := pNode^;
END_METHOD

METHOD FB_init : BOOL
VAR_INPUT
	bInitRetains : BOOL; // if TRUE, the retain variables are initialized (warm start / cold start)
	bInCopyCode : BOOL;  // if TRUE, the instance afterwards gets moved into the copy code (online change)
END_VAR
AddInput('in1',THIS^.in1);
AddInput('in2',THIS^.in2);
AddOutput('out', THIS^.out);
END_METHOD

METHOD PROTECTED OnExecute
VAR
END_VAR
out.Value := in1.Value * in2.Value;
END_METHOD

END_FUNCTION_BLOCK

// ---- Core/Nodes/MUL/MUL_LINT.TcPOU
{attribute 'linkalways'} 
{attribute 'no_explicit_call' := 'This FB is a CLASS and must be accessed using methods or properties'}
{attribute 'enable_dynamic_creation'}
FUNCTION_BLOCK FINAL MUL_LINT EXTENDS Node
VAR
	in1 : _LINT(0);
	in2 : _LINT(0);
	out : _LINT(0);
END_VAR

METHOD PUBLIC Clone : I_Node
VAR
	pNode : POINTER TO MUL_LINT;
END_VAR
pNode := __NEW(MUL_LINT);
Clone := pNode^;
END_METHOD

METHOD FB_init : BOOL
VAR_INPUT
	bInitRetains : BOOL; // if TRUE, the retain variables are initialized (warm start / cold start)
	bInCopyCode : BOOL;  // if TRUE, the instance afterwards gets moved into the copy code (online change)
END_VAR
AddInput('in1',THIS^.in1);
AddInput('in2',THIS^.in2);
AddOutput('out', THIS^.out);
END_METHOD

METHOD PROTECTED OnExecute
VAR
END_VAR
out.Value := in1.Value * in2.Value;
END_METHOD

END_FUNCTION_BLOCK

// ---- Core/Nodes/MUL/MUL_LREAL.TcPOU
{attribute 'linkalways'} 
{attribute 'no_explicit_call' := 'This FB is a CLASS and must be accessed using methods or properties'}
{attribute 'enable_dynamic_creation'}
FUNCTION_BLOCK FINAL MUL_LREAL EXTENDS Node
VAR
	in1 : _LREAL(0.0);
	in2 : _LREAL(0.0);
	out : _LREAL(0.0);
END_VAR

METHOD PUBLIC Clone : I_Node
VAR
	pNode : POINTER TO MUL_LREAL;
END_VAR
pNode := __NEW(MUL_LREAL);
Clone := pNode^;
END_METHOD

METHOD FB_init : BOOL
VAR_INPUT
	bInitRetains : BOOL; // if TRUE, the retain variables are initialized (warm start / cold start)
	bInCopyCode : BOOL;  // if TRUE, the instance afterwards gets moved into the copy code (online change)
END_VAR
AddInput('in1',THIS^.in1);
AddInput('in2',THIS^.in2);
AddOutput('out', THIS^.out);
END_METHOD

METHOD PROTECTED OnExecute
VAR
END_VAR
out.Value := in1.Value * in2.Value;
END_METHOD

END_FUNCTION_BLOCK

// ---- Core/Nodes/MUL/MUL_LWORD.TcPOU
{attribute 'linkalways'} 
{attribute 'no_explicit_call' := 'This FB is a CLASS and must be accessed using methods or properties'}
{attribute 'enable_dynamic_creation'}
FUNCTION_BLOCK FINAL MUL_LWORD EXTENDS Node
VAR
	in1 : _LWORD(0);
	in2 : _LWORD(0);
	out : _LWORD(0);
END_VAR

METHOD PUBLIC Clone : I_Node
VAR
	pNode : POINTER TO MUL_LWORD;
END_VAR
pNode := __NEW(MUL_LWORD);
Clone := pNode^;
END_METHOD

METHOD FB_init : BOOL
VAR_INPUT
	bInitRetains : BOOL; // if TRUE, the retain variables are initialized (warm start / cold start)
	bInCopyCode : BOOL;  // if TRUE, the instance afterwards gets moved into the copy code (online change)
END_VAR
AddInput('in1',THIS^.in1);
AddInput('in2',THIS^.in2);
AddOutput('out', THIS^.out);
END_METHOD

METHOD PROTECTED OnExecute
VAR
END_VAR
out.Value := in1.Value * in2.Value;
END_METHOD

END_FUNCTION_BLOCK

// ---- Core/Nodes/MUL/MUL_REAL.TcPOU
{attribute 'linkalways'} 
{attribute 'no_explicit_call' := 'This FB is a CLASS and must be accessed using methods or properties'}
{attribute 'enable_dynamic_creation'}
FUNCTION_BLOCK FINAL MUL_REAL EXTENDS Node
VAR
	in1 : _REAL(0.0);
	in2 : _REAL(0.0);
	out : _REAL(0.0);
END_VAR

METHOD PUBLIC Clone : I_Node
VAR
	pNode : POINTER TO MUL_REAL;
END_VAR
pNode := __NEW(MUL_REAL);
Clone := pNode^;
END_METHOD

METHOD FB_init : BOOL
VAR_INPUT
	bInitRetains : BOOL; // if TRUE, the retain variables are initialized (warm start / cold start)
	bInCopyCode : BOOL;  // if TRUE, the instance afterwards gets moved into the copy code (online change)
END_VAR
AddInput('in1',THIS^.in1);
AddInput('in2',THIS^.in2);
AddOutput('out', THIS^.out);
END_METHOD

METHOD PROTECTED OnExecute
VAR
END_VAR
out.Value := in1.Value * in2.Value;
END_METHOD

END_FUNCTION_BLOCK

// ---- Core/Nodes/MUL/MUL_SINT.TcPOU
{attribute 'linkalways'} 
{attribute 'no_explicit_call' := 'This FB is a CLASS and must be accessed using methods or properties'}
{attribute 'enable_dynamic_creation'}
FUNCTION_BLOCK FINAL MUL_SINT EXTENDS Node
VAR
	in1 : _SINT(0);
	in2 : _SINT(0);
	out : _SINT(0);
END_VAR

METHOD PUBLIC Clone : I_Node
VAR
	pNode : POINTER TO MUL_SINT;
END_VAR
pNode := __NEW(MUL_SINT);
Clone := pNode^;
END_METHOD

METHOD FB_init : BOOL
VAR_INPUT
	bInitRetains : BOOL; // if TRUE, the retain variables are initialized (warm start / cold start)
	bInCopyCode : BOOL;  // if TRUE, the instance afterwards gets moved into the copy code (online change)
END_VAR
AddInput('in1',THIS^.in1);
AddInput('in2',THIS^.in2);
AddOutput('out', THIS^.out);
END_METHOD

METHOD PROTECTED OnExecute
VAR
END_VAR
out.Value := in1.Value * in2.Value;
END_METHOD

END_FUNCTION_BLOCK

// ---- Core/Nodes/MUL/MUL_UDINT.TcPOU
{attribute 'linkalways'} 
{attribute 'no_explicit_call' := 'This FB is a CLASS and must be accessed using methods or properties'}
{attribute 'enable_dynamic_creation'}
FUNCTION_BLOCK FINAL MUL_UDINT EXTENDS Node
VAR
	in1 : _UDINT(0);
	in2 : _UDINT(0);
	out : _UDINT(0);
END_VAR

METHOD PUBLIC Clone : I_Node
VAR
	pNode : POINTER TO MUL_UDINT;
END_VAR
pNode := __NEW(MUL_UDINT);
Clone := pNode^;
END_METHOD

METHOD FB_init : BOOL
VAR_INPUT
	bInitRetains : BOOL; // if TRUE, the retain variables are initialized (warm start / cold start)
	bInCopyCode : BOOL;  // if TRUE, the instance afterwards gets moved into the copy code (online change)
END_VAR
AddInput('in1',THIS^.in1);
AddInput('in2',THIS^.in2);
AddOutput('out', THIS^.out);
END_METHOD

METHOD PROTECTED OnExecute
VAR
END_VAR
out.Value := in1.Value * in2.Value;
END_METHOD

END_FUNCTION_BLOCK

// ---- Core/Nodes/MUL/MUL_UINT.TcPOU
{attribute 'linkalways'} 
{attribute 'no_explicit_call' := 'This FB is a CLASS and must be accessed using methods or properties'}
{attribute 'enable_dynamic_creation'}
FUNCTION_BLOCK FINAL MUL_UINT EXTENDS Node
VAR
	in1 : _UINT(0);
	in2 : _UINT(0);
	out : _UINT(0);
END_VAR

METHOD PUBLIC Clone : I_Node
VAR
	pNode : POINTER TO MUL_UINT;
END_VAR
pNode := __NEW(MUL_UINT);
Clone := pNode^;
END_METHOD

METHOD FB_init : BOOL
VAR_INPUT
	bInitRetains : BOOL; // if TRUE, the retain variables are initialized (warm start / cold start)
	bInCopyCode : BOOL;  // if TRUE, the instance afterwards gets moved into the copy code (online change)
END_VAR
AddInput('in1',THIS^.in1);
AddInput('in2',THIS^.in2);
AddOutput('out', THIS^.out);
END_METHOD

METHOD PROTECTED OnExecute
VAR
END_VAR
out.Value := in1.Value * in2.Value;
END_METHOD

END_FUNCTION_BLOCK

// ---- Core/Nodes/MUL/MUL_ULINT.TcPOU
{attribute 'linkalways'} 
{attribute 'no_explicit_call' := 'This FB is a CLASS and must be accessed using methods or properties'}
{attribute 'enable_dynamic_creation'}
FUNCTION_BLOCK FINAL MUL_ULINT EXTENDS Node
VAR
	in1 : _ULINT(0);
	in2 : _ULINT(0);
	out : _ULINT(0);
END_VAR

METHOD PUBLIC Clone : I_Node
VAR
	pNode : POINTER TO MUL_ULINT;
END_VAR
pNode := __NEW(MUL_ULINT);
Clone := pNode^;
END_METHOD

METHOD FB_init : BOOL
VAR_INPUT
	bInitRetains : BOOL; // if TRUE, the retain variables are initialized (warm start / cold start)
	bInCopyCode : BOOL;  // if TRUE, the instance afterwards gets moved into the copy code (online change)
END_VAR
AddInput('in1',THIS^.in1);
AddInput('in2',THIS^.in2);
AddOutput('out', THIS^.out);
END_METHOD

METHOD PROTECTED OnExecute
VAR
END_VAR
out.Value := in1.Value * in2.Value;
END_METHOD

END_FUNCTION_BLOCK

// ---- Core/Nodes/MUL/MUL_USINT.TcPOU
{attribute 'linkalways'} 
{attribute 'no_explicit_call' := 'This FB is a CLASS and must be accessed using methods or properties'}
{attribute 'enable_dynamic_creation'}
FUNCTION_BLOCK FINAL MUL_USINT EXTENDS Node
VAR
	in1 : _USINT(0);
	in2 : _USINT(0);
	out : _USINT(0);
END_VAR

METHOD PUBLIC Clone : I_Node
VAR
	pNode : POINTER TO MUL_USINT;
END_VAR
pNode := __NEW(MUL_USINT);
Clone := pNode^;
END_METHOD

METHOD FB_init : BOOL
VAR_INPUT
	bInitRetains : BOOL; // if TRUE, the retain variables are initialized (warm start / cold start)
	bInCopyCode : BOOL;  // if TRUE, the instance afterwards gets moved into the copy code (online change)
END_VAR
AddInput('in1',THIS^.in1);
AddInput('in2',THIS^.in2);
AddOutput('out', THIS^.out);
END_METHOD

METHOD PROTECTED OnExecute
VAR
END_VAR
out.Value := in1.Value * in2.Value;
END_METHOD

END_FUNCTION_BLOCK

// ---- Core/Nodes/MUL/MUL_WORD.TcPOU
{attribute 'linkalways'} 
{attribute 'no_explicit_call' := 'This FB is a CLASS and must be accessed using methods or properties'}
{attribute 'enable_dynamic_creation'}
FUNCTION_BLOCK FINAL MUL_WORD EXTENDS Node
VAR
	in1 : _WORD(0);
	in2 : _WORD(0);
	out : _WORD(0);
END_VAR

METHOD PUBLIC Clone : I_Node
VAR
	pNode : POINTER TO MUL_WORD;
END_VAR
pNode := __NEW(MUL_WORD);
Clone := pNode^;
END_METHOD

METHOD FB_init : BOOL
VAR_INPUT
	bInitRetains : BOOL; // if TRUE, the retain variables are initialized (warm start / cold start)
	bInCopyCode : BOOL;  // if TRUE, the instance afterwards gets moved into the copy code (online change)
END_VAR
AddInput('in1',THIS^.in1);
AddInput('in2',THIS^.in2);
AddOutput('out', THIS^.out);
END_METHOD

METHOD PROTECTED OnExecute
VAR
END_VAR
out.Value := in1.Value - in2.Value;
END_METHOD

END_FUNCTION_BLOCK

// ---- Core/Nodes/DIV/DIV_BYTE.TcPOU
{attribute 'linkalways'} 
{attribute 'no_explicit_call' := 'This FB is a CLASS and must be accessed using methods or properties'}
{attribute 'enable_dynamic_creation'}
FUNCTION_BLOCK FINAL DIV_BYTE EXTENDS Node
VAR
	in1 : _BYTE(0);
	in2 : _BYTE(0);
	out : _BYTE(0);
	div0 : _BOOL(FALSE);
END_VAR

METHOD PUBLIC Clone : I_Node
VAR
	pNode : POINTER TO DIV_BYTE;
END_VAR
pNode := __NEW(DIV_BYTE);
Clone := pNode^;
END_METHOD

METHOD FB_init : BOOL
VAR_INPUT
	bInitRetains : BOOL; // if TRUE, the retain variables are initialized (warm start / cold start)
	bInCopyCode : BOOL;  // if TRUE, the instance afterwards gets moved into the copy code (online change)
END_VAR
AddInput('in1',THIS^.in1);
AddInput('in2',THIS^.in2);
AddOutput('out', THIS^.out);
AddOutput('div0', THIS^.div0);
END_METHOD

METHOD PROTECTED OnExecute
VAR
END_VAR
IF in2.Value = 0 THEN
	div0.Value := TRUE;
	RETURN;
END_IF

out.Value := in1.Value / in2.Value;
div0.Value := FALSE;
END_METHOD

END_FUNCTION_BLOCK

// ---- Core/Nodes/DIV/DIV_DINT.TcPOU
{attribute 'linkalways'} 
{attribute 'no_explicit_call' := 'This FB is a CLASS and must be accessed using methods or properties'}
{attribute 'enable_dynamic_creation'}
FUNCTION_BLOCK FINAL DIV_DINT EXTENDS Node
VAR
	in1 : _DINT(0);
	in2 : _DINT(0);
	out : _DINT(0);
	div0 : _BOOL(FALSE);
END_VAR

METHOD PUBLIC Clone : I_Node
VAR
	pNode : POINTER TO DIV_DINT;
END_VAR
pNode := __NEW(DIV_DINT);
Clone := pNode^;
END_METHOD

METHOD FB_init : BOOL
VAR_INPUT
	bInitRetains : BOOL; // if TRUE, the retain variables are initialized (warm start / cold start)
	bInCopyCode : BOOL;  // if TRUE, the instance afterwards gets moved into the copy code (online change)
END_VAR
AddInput('in1',THIS^.in1);
AddInput('in2',THIS^.in2);
AddOutput('out', THIS^.out);
AddOutput('div0', THIS^.div0);
END_METHOD

METHOD PROTECTED OnExecute
VAR
END_VAR
IF in2.Value = 0 THEN
	div0.Value := TRUE;
	RETURN;
END_IF

out.Value := in1.Value / in2.Value;
div0.Value := FALSE;
END_METHOD

END_FUNCTION_BLOCK

// ---- Core/Nodes/DIV/DIV_DWORD.TcPOU
{attribute 'linkalways'} 
{attribute 'no_explicit_call' := 'This FB is a CLASS and must be accessed using methods or properties'}
{attribute 'enable_dynamic_creation'}
FUNCTION_BLOCK FINAL DIV_DWORD EXTENDS Node
VAR
	in1 : _DWORD(0);
	in2 : _DWORD(0);
	out : _DWORD(0);
	div0 : _BOOL(FALSE);
END_VAR

METHOD PUBLIC Clone : I_Node
VAR
	pNode : POINTER TO DIV_DWORD;
END_VAR
pNode := __NEW(DIV_DWORD);
Clone := pNode^;
END_METHOD

METHOD FB_init : BOOL
VAR_INPUT
	bInitRetains : BOOL; // if TRUE, the retain variables are initialized (warm start / cold start)
	bInCopyCode : BOOL;  // if TRUE, the instance afterwards gets moved into the copy code (online change)
END_VAR
AddInput('in1',THIS^.in1);
AddInput('in2',THIS^.in2);
AddOutput('out', THIS^.out);
AddOutput('div0', THIS^.div0);
END_METHOD

METHOD PROTECTED OnExecute
VAR
END_VAR
IF in2.Value = 0 THEN
	div0.Value := TRUE;
	RETURN;
END_IF

out.Value := in1.Value / in2.Value;
div0.Value := FALSE;
END_METHOD

END_FUNCTION_BLOCK

// ---- Core/Nodes/DIV/DIV_INT.TcPOU
{attribute 'linkalways'} 
{attribute 'no_explicit_call' := 'This FB is a CLASS and must be accessed using methods or properties'}
{attribute 'enable_dynamic_creation'}
FUNCTION_BLOCK FINAL DIV_INT EXTENDS Node
VAR
	in1 : _INT(0);
	in2 : _INT(0);
	out : _INT(0);
	div0 : _BOOL(FALSE);
END_VAR

METHOD PUBLIC Clone : I_Node
VAR
	pNode : POINTER TO DIV_INT;
END_VAR
pNode := __NEW(DIV_INT);
Clone := pNode^;
END_METHOD

METHOD FB_init : BOOL
VAR_INPUT
	bInitRetains : BOOL; // if TRUE, the retain variables are initialized (warm start / cold start)
	bInCopyCode : BOOL;  // if TRUE, the instance afterwards gets moved into the copy code (online change)
END_VAR
AddInput('in1',THIS^.in1);
AddInput('in2',THIS^.in2);
AddOutput('out', THIS^.out);
AddOutput('div0', THIS^.div0);
END_METHOD

METHOD PROTECTED OnExecute
VAR
END_VAR
IF in2.Value = 0 THEN
	div0.Value := TRUE;
	RETURN;
END_IF

out.Value := in1.Value / in2.Value;
div0.Value := FALSE;
END_METHOD

END_FUNCTION_BLOCK

// ---- Core/Nodes/DIV/DIV_LINT.TcPOU
{attribute 'linkalways'} 
{attribute 'no_explicit_call' := 'This FB is a CLASS and must be accessed using methods or properties'}
{attribute 'enable_dynamic_creation'}
FUNCTION_BLOCK FINAL DIV_LINT EXTENDS Node
VAR
	in1 : _LINT(0);
	in2 : _LINT(0);
	out : _LINT(0);
	div0 : _BOOL(FALSE);
END_VAR

METHOD PUBLIC Clone : I_Node
VAR
	pNode : POINTER TO DIV_LINT;
END_VAR
pNode := __NEW(DIV_LINT);
Clone := pNode^;
END_METHOD

METHOD FB_init : BOOL
VAR_INPUT
	bInitRetains : BOOL; // if TRUE, the retain variables are initialized (warm start / cold start)
	bInCopyCode : BOOL;  // if TRUE, the instance afterwards gets moved into the copy code (online change)
END_VAR
AddInput('in1',THIS^.in1);
AddInput('in2',THIS^.in2);
AddOutput('out', THIS^.out);
AddOutput('div0', THIS^.div0);
END_METHOD

METHOD PROTECTED OnExecute
VAR
END_VAR
IF in2.Value = 0 THEN
	div0.Value := TRUE;
	RETURN;
END_IF

out.Value := in1.Value / in2.Value;
div0.Value := FALSE;
END_METHOD

END_FUNCTION_BLOCK

// ---- Core/Nodes/DIV/DIV_LREAL.TcPOU
{attribute 'linkalways'} 
{attribute 'no_explicit_call' := 'This FB is a CLASS and must be accessed using methods or properties'}
{attribute 'enable_dynamic_creation'}
FUNCTION_BLOCK FINAL DIV_LREAL EXTENDS Node
VAR
	in1 : _LREAL(0.0);
	in2 : _LREAL(0.0);
	out : _LREAL(0.0);
	div0 : _BOOL(FALSE);
END_VAR

METHOD PUBLIC Clone : I_Node
VAR
	pNode : POINTER TO DIV_LREAL;
END_VAR
pNode := __NEW(DIV_LREAL);
Clone := pNode^;
END_METHOD

METHOD FB_init : BOOL
VAR_INPUT
	bInitRetains : BOOL; // if TRUE, the retain variables are initialized (warm start / cold start)
	bInCopyCode : BOOL;  // if TRUE, the instance afterwards gets moved into the copy code (online change)
END_VAR
AddInput('in1',THIS^.in1);
AddInput('in2',THIS^.in2);
AddOutput('out', THIS^.out);
AddOutput('div0', THIS^.div0);
END_METHOD

METHOD PROTECTED OnExecute
VAR
END_VAR
IF in2.Value = 0 THEN
	div0.Value := TRUE;
	RETURN;
END_IF

out.Value := in1.Value / in2.Value;
div0.Value := FALSE;
END_METHOD

END_FUNCTION_BLOCK

// ---- Core/Nodes/DIV/DIV_LWORD.TcPOU
{attribute 'linkalways'} 
{attribute 'no_explicit_call' := 'This FB is a CLASS and must be accessed using methods or properties'}
{attribute 'enable_dynamic_creation'}
FUNCTION_BLOCK FINAL DIV_LWORD EXTENDS Node
VAR
	in1 : _LWORD(0);
	in2 : _LWORD(0);
	out : _LWORD(0);
	div0 : _BOOL(FALSE);
END_VAR

METHOD PUBLIC Clone : I_Node
VAR
	pNode : POINTER TO DIV_LWORD;
END_VAR
pNode := __NEW(DIV_LWORD);
Clone := pNode^;
END_METHOD

METHOD FB_init : BOOL
VAR_INPUT
	bInitRetains : BOOL; // if TRUE, the retain variables are initialized (warm start / cold start)
	bInCopyCode : BOOL;  // if TRUE, the instance afterwards gets moved into the copy code (online change)
END_VAR
AddInput('in1',THIS^.in1);
AddInput('in2',THIS^.in2);
AddOutput('out', THIS^.out);
AddOutput('div0', THIS^.div0);
END_METHOD

METHOD PROTECTED OnExecute
VAR
END_VAR
IF in2.Value = 0 THEN
	div0.Value := TRUE;
	RETURN;
END_IF

out.Value := in1.Value / in2.Value;
div0.Value := FALSE;
END_METHOD

END_FUNCTION_BLOCK

// ---- Core/Nodes/DIV/DIV_REAL.TcPOU
{attribute 'linkalways'} 
{attribute 'no_explicit_call' := 'This FB is a CLASS and must be accessed using methods or properties'}
{attribute 'enable_dynamic_creation'}
FUNCTION_BLOCK FINAL DIV_REAL EXTENDS Node
VAR
	in1 : _REAL(0.0);
	in2 : _REAL(0.0);
	out : _REAL(0.0);
	div0 : _BOOL(FALSE);
END_VAR

METHOD PUBLIC Clone : I_Node
VAR
	pNode : POINTER TO DIV_REAL;
END_VAR
pNode := __NEW(DIV_REAL);
Clone := pNode^;
END_METHOD

METHOD FB_init : BOOL
VAR_INPUT
	bInitRetains : BOOL; // if TRUE, the retain variables are initialized (warm start / cold start)
	bInCopyCode : BOOL;  // if TRUE, the instance afterwards gets moved into the copy code (online change)
END_VAR
AddInput('in1',THIS^.in1);
AddInput('in2',THIS^.in2);
AddOutput('out', THIS^.out);
AddOutput('div0', THIS^.div0);
END_METHOD

METHOD PROTECTED OnExecute
VAR
END_VAR
IF in2.Value = 0 THEN
	div0.Value := TRUE;
	RETURN;
END_IF

out.Value := in1.Value / in2.Value;
div0.Value := FALSE;
END_METHOD

END_FUNCTION_BLOCK

// ---- Core/Nodes/DIV/DIV_SINT.TcPOU
{attribute 'linkalways'} 
{attribute 'no_explicit_call' := 'This FB is a CLASS and must be accessed using methods or properties'}
{attribute 'enable_dynamic_creation'}
FUNCTION_BLOCK FINAL DIV_SINT EXTENDS Node
VAR
	in1 : _SINT(0);
	in2 : _SINT(0);
	out : _SINT(0);
	div0 : _BOOL(FALSE);
END_VAR

METHOD PUBLIC Clone : I_Node
VAR
	pNode : POINTER TO DIV_SINT;
END_VAR
pNode := __NEW(DIV_SINT);
Clone := pNode^;
END_METHOD

METHOD FB_init : BOOL
VAR_INPUT
	bInitRetains : BOOL; // if TRUE, the retain variables are initialized (warm start / cold start)
	bInCopyCode : BOOL;  // if TRUE, the instance afterwards gets moved into the copy code (online change)
END_VAR
AddInput('in1',THIS^.in1);
AddInput('in2',THIS^.in2);
AddOutput('out', THIS^.out);
AddOutput('div0', THIS^.div0);
END_METHOD

METHOD PROTECTED OnExecute
VAR
END_VAR
IF in2.Value = 0 THEN
	div0.Value := TRUE;
	RETURN;
END_IF

out.Value := in1.Value / in2.Value;
div0.Value := FALSE;
END_METHOD

END_FUNCTION_BLOCK

// ---- Core/Nodes/DIV/DIV_UDINT.TcPOU
{attribute 'linkalways'} 
{attribute 'no_explicit_call' := 'This FB is a CLASS and must be accessed using methods or properties'}
{attribute 'enable_dynamic_creation'}
FUNCTION_BLOCK FINAL DIV_UDINT EXTENDS Node
VAR
	in1 : _UDINT(0);
	in2 : _UDINT(0);
	out : _UDINT(0);
	div0 : _BOOL(FALSE);
END_VAR

METHOD PUBLIC Clone : I_Node
VAR
	pNode : POINTER TO DIV_UDINT;
END_VAR
pNode := __NEW(DIV_UDINT);
Clone := pNode^;
END_METHOD

METHOD FB_init : BOOL
VAR_INPUT
	bInitRetains : BOOL; // if TRUE, the retain variables are initialized (warm start / cold start)
	bInCopyCode : BOOL;  // if TRUE, the instance afterwards gets moved into the copy code (online change)
END_VAR
AddInput('in1',THIS^.in1);
AddInput('in2',THIS^.in2);
AddOutput('out', THIS^.out);
AddOutput('div0', THIS^.div0);
END_METHOD

METHOD PROTECTED OnExecute
VAR
END_VAR
IF in2.Value = 0 THEN
	div0.Value := TRUE;
	RETURN;
END_IF

out.Value := in1.Value / in2.Value;
div0.Value := FALSE;
END_METHOD

END_FUNCTION_BLOCK

// ---- Core/Nodes/DIV/DIV_UINT.TcPOU
{attribute 'linkalways'} 
{attribute 'no_explicit_call' := 'This FB is a CLASS and must be accessed using methods or properties'}
{attribute 'enable_dynamic_creation'}
FUNCTION_BLOCK FINAL DIV_UINT EXTENDS Node
VAR
	in1 : _UINT(0);
	in2 : _UINT(0);
	out : _UINT(0);
	div0 : _BOOL(FALSE);
END_VAR

METHOD PUBLIC Clone : I_Node
VAR
	pNode : POINTER TO DIV_UINT;
END_VAR
pNode := __NEW(DIV_UINT);
Clone := pNode^;
END_METHOD

METHOD FB_init : BOOL
VAR_INPUT
	bInitRetains : BOOL; // if TRUE, the retain variables are initialized (warm start / cold start)
	bInCopyCode : BOOL;  // if TRUE, the instance afterwards gets moved into the copy code (online change)
END_VAR
AddInput('in1',THIS^.in1);
AddInput('in2',THIS^.in2);
AddOutput('out', THIS^.out);
AddOutput('div0', THIS^.div0);
END_METHOD

METHOD PROTECTED OnExecute
VAR
END_VAR
IF in2.Value = 0 THEN
	div0.Value := TRUE;
	RETURN;
END_IF

out.Value := in1.Value / in2.Value;
div0.Value := FALSE;
END_METHOD

END_FUNCTION_BLOCK

// ---- Core/Nodes/DIV/DIV_ULINT.TcPOU
{attribute 'linkalways'} 
{attribute 'no_explicit_call' := 'This FB is a CLASS and must be accessed using methods or properties'}
{attribute 'enable_dynamic_creation'}
FUNCTION_BLOCK FINAL DIV_ULINT EXTENDS Node
VAR
	in1 : _ULINT(0);
	in2 : _ULINT(0);
	out : _ULINT(0);
	div0 : _BOOL(FALSE);
END_VAR

METHOD PUBLIC Clone : I_Node
VAR
	pNode : POINTER TO DIV_ULINT;
END_VAR
pNode := __NEW(DIV_ULINT);
Clone := pNode^;
END_METHOD

METHOD FB_init : BOOL
VAR_INPUT
	bInitRetains : BOOL; // if TRUE, the retain variables are initialized (warm start / cold start)
	bInCopyCode : BOOL;  // if TRUE, the instance afterwards gets moved into the copy code (online change)
END_VAR
AddInput('in1',THIS^.in1);
AddInput('in2',THIS^.in2);
AddOutput('out', THIS^.out);
AddOutput('div0', THIS^.div0);
END_METHOD

METHOD PROTECTED OnExecute
VAR
END_VAR
IF in2.Value = 0 THEN
	div0.Value := TRUE;
	RETURN;
END_IF

out.Value := in1.Value / in2.Value;
div0.Value := FALSE;
END_METHOD

END_FUNCTION_BLOCK

// ---- Core/Nodes/DIV/DIV_USINT.TcPOU
{attribute 'linkalways'} 
{attribute 'no_explicit_call' := 'This FB is a CLASS and must be accessed using methods or properties'}
{attribute 'enable_dynamic_creation'}
FUNCTION_BLOCK FINAL DIV_USINT EXTENDS Node
VAR
	in1 : _USINT(0);
	in2 : _USINT(0);
	out : _USINT(0);
	div0 : _BOOL(FALSE);
END_VAR

METHOD PUBLIC Clone : I_Node
VAR
	pNode : POINTER TO DIV_USINT;
END_VAR
pNode := __NEW(DIV_USINT);
Clone := pNode^;
END_METHOD

METHOD FB_init : BOOL
VAR_INPUT
	bInitRetains : BOOL; // if TRUE, the retain variables are initialized (warm start / cold start)
	bInCopyCode : BOOL;  // if TRUE, the instance afterwards gets moved into the copy code (online change)
END_VAR
AddInput('in1',THIS^.in1);
AddInput('in2',THIS^.in2);
AddOutput('out', THIS^.out);
AddOutput('div0', THIS^.div0);
END_METHOD

METHOD PROTECTED OnExecute
VAR
END_VAR
IF in2.Value = 0 THEN
	div0.Value := TRUE;
	RETURN;
END_IF

out.Value := in1.Value / in2.Value;
div0.Value := FALSE;
END_METHOD

END_FUNCTION_BLOCK

// ---- Core/Nodes/DIV/DIV_WORD.TcPOU
{attribute 'linkalways'} 
{attribute 'no_explicit_call' := 'This FB is a CLASS and must be accessed using methods or properties'}
{attribute 'enable_dynamic_creation'}
FUNCTION_BLOCK FINAL DIV_WORD EXTENDS Node
VAR
	in1 : _WORD(0);
	in2 : _WORD(0);
	out : _WORD(0);
	div0 : _BOOL(FALSE);
END_VAR

METHOD PUBLIC Clone : I_Node
VAR
	pNode : POINTER TO DIV_WORD;
END_VAR
pNode := __NEW(DIV_WORD);
Clone := pNode^;
END_METHOD

METHOD FB_init : BOOL
VAR_INPUT
	bInitRetains : BOOL; // if TRUE, the retain variables are initialized (warm start / cold start)
	bInCopyCode : BOOL;  // if TRUE, the instance afterwards gets moved into the copy code (online change)
END_VAR
AddInput('in1',THIS^.in1);
AddInput('in2',THIS^.in2);
AddOutput('out', THIS^.out);
AddOutput('div0', THIS^.div0);
END_METHOD

METHOD PROTECTED OnExecute
VAR
END_VAR
IF in2.Value = 0 THEN
	div0.Value := TRUE;
	RETURN;
END_IF

out.Value := in1.Value / in2.Value;
div0.Value := FALSE;
END_METHOD

END_FUNCTION_BLOCK

// ---- Core/Nodes/MOD/MOD_BYTE.TcPOU
{attribute 'linkalways'} 
{attribute 'no_explicit_call' := 'This FB is a CLASS and must be accessed using methods or properties'}
{attribute 'enable_dynamic_creation'}
FUNCTION_BLOCK FINAL MOD_BYTE EXTENDS Node
VAR
	in1 : _BYTE(0);
	in2 : _BYTE(0);
	out : _BYTE(0);
END_VAR

METHOD PUBLIC Clone : I_Node
VAR
	pNode : POINTER TO MOD_BYTE;
END_VAR
pNode := __NEW(MOD_BYTE);
Clone := pNode^;
END_METHOD

METHOD FB_init : BOOL
VAR_INPUT
	bInitRetains : BOOL; // if TRUE, the retain variables are initialized (warm start / cold start)
	bInCopyCode : BOOL;  // if TRUE, the instance afterwards gets moved into the copy code (online change)
END_VAR
AddInput('in1',THIS^.in1);
AddInput('in2',THIS^.in2);
AddOutput('out', THIS^.out);
END_METHOD

METHOD PROTECTED OnExecute
VAR
END_VAR
out.Value := in1.Value MOD in2.Value;
END_METHOD

END_FUNCTION_BLOCK

// ---- Core/Nodes/MOD/MOD_DINT.TcPOU
{attribute 'linkalways'} 
{attribute 'no_explicit_call' := 'This FB is a CLASS and must be accessed using methods or properties'}
{attribute 'enable_dynamic_creation'}
FUNCTION_BLOCK FINAL MOD_DINT EXTENDS Node
VAR
	in1 : _DINT(0);
	in2 : _DINT(0);
	out : _DINT(0);
END_VAR

METHOD PUBLIC Clone : I_Node
VAR
	pNode : POINTER TO MOD_DINT;
END_VAR
pNode := __NEW(MOD_DINT);
Clone := pNode^;
END_METHOD

METHOD FB_init : BOOL
VAR_INPUT
	bInitRetains : BOOL; // if TRUE, the retain variables are initialized (warm start / cold start)
	bInCopyCode : BOOL;  // if TRUE, the instance afterwards gets moved into the copy code (online change)
END_VAR
AddInput('in1',THIS^.in1);
AddInput('in2',THIS^.in2);
AddOutput('out', THIS^.out);
END_METHOD

METHOD PROTECTED OnExecute
VAR
END_VAR
out.Value := in1.Value MOD in2.Value;
END_METHOD

END_FUNCTION_BLOCK

// ---- Core/Nodes/MOD/MOD_DWORD.TcPOU
{attribute 'linkalways'} 
{attribute 'no_explicit_call' := 'This FB is a CLASS and must be accessed using methods or properties'}
{attribute 'enable_dynamic_creation'}
FUNCTION_BLOCK FINAL MOD_DWORD EXTENDS Node
VAR
	in1 : _DWORD(0);
	in2 : _DWORD(0);
	out : _DWORD(0);
END_VAR

METHOD PUBLIC Clone : I_Node
VAR
	pNode : POINTER TO MOD_DWORD;
END_VAR
pNode := __NEW(MOD_DWORD);
Clone := pNode^;
END_METHOD

METHOD FB_init : BOOL
VAR_INPUT
	bInitRetains : BOOL; // if TRUE, the retain variables are initialized (warm start / cold start)
	bInCopyCode : BOOL;  // if TRUE, the instance afterwards gets moved into the copy code (online change)
END_VAR
AddInput('in1',THIS^.in1);
AddInput('in2',THIS^.in2);
AddOutput('out', THIS^.out);
END_METHOD

METHOD PROTECTED OnExecute
VAR
END_VAR
out.Value := in1.Value MOD in2.Value;
END_METHOD

END_FUNCTION_BLOCK

// ---- Core/Nodes/MOD/MOD_INT.TcPOU
{attribute 'linkalways'} 
{attribute 'no_explicit_call' := 'This FB is a CLASS and must be accessed using methods or properties'}
{attribute 'enable_dynamic_creation'}
FUNCTION_BLOCK FINAL MOD_INT EXTENDS Node
VAR
	in1 : _INT(0);
	in2 : _INT(0);
	out : _INT(0);
END_VAR

METHOD PUBLIC Clone : I_Node
VAR
	pNode : POINTER TO MOD_INT;
END_VAR
pNode := __NEW(MOD_INT);
Clone := pNode^;
END_METHOD

METHOD FB_init : BOOL
VAR_INPUT
	bInitRetains : BOOL; // if TRUE, the retain variables are initialized (warm start / cold start)
	bInCopyCode : BOOL;  // if TRUE, the instance afterwards gets moved into the copy code (online change)
END_VAR
AddInput('in1',THIS^.in1);
AddInput('in2',THIS^.in2);
AddOutput('out', THIS^.out);
END_METHOD

METHOD PROTECTED OnExecute
VAR
END_VAR
out.Value := in1.Value MOD in2.Value;
END_METHOD

END_FUNCTION_BLOCK

// ---- Core/Nodes/MOD/MOD_LINT.TcPOU
{attribute 'linkalways'} 
{attribute 'no_explicit_call' := 'This FB is a CLASS and must be accessed using methods or properties'}
{attribute 'enable_dynamic_creation'}
FUNCTION_BLOCK FINAL MOD_LINT EXTENDS Node
VAR
	in1 : _LINT(0);
	in2 : _LINT(0);
	out : _LINT(0);
END_VAR

METHOD PUBLIC Clone : I_Node
VAR
	pNode : POINTER TO MOD_LINT;
END_VAR
pNode := __NEW(MOD_LINT);
Clone := pNode^;
END_METHOD

METHOD FB_init : BOOL
VAR_INPUT
	bInitRetains : BOOL; // if TRUE, the retain variables are initialized (warm start / cold start)
	bInCopyCode : BOOL;  // if TRUE, the instance afterwards gets moved into the copy code (online change)
END_VAR
AddInput('in1',THIS^.in1);
AddInput('in2',THIS^.in2);
AddOutput('out', THIS^.out);
END_METHOD

METHOD PROTECTED OnExecute
VAR
END_VAR
out.Value := in1.Value MOD in2.Value;
END_METHOD

END_FUNCTION_BLOCK

// ---- Core/Nodes/MOD/MOD_LREAL.TcPOU
{attribute 'linkalways'} 
{attribute 'no_explicit_call' := 'This FB is a CLASS and must be accessed using methods or properties'}
{attribute 'enable_dynamic_creation'}
FUNCTION_BLOCK FINAL MOD_LREAL EXTENDS Node
VAR
	in1 : _LREAL(0.0);
	in2 : _LREAL(0.0);
	out : _LREAL(0.0);
END_VAR

METHOD PUBLIC Clone : I_Node
VAR
	pNode : POINTER TO MOD_LREAL;
END_VAR
pNode := __NEW(MOD_LREAL);
Clone := pNode^;
END_METHOD

METHOD FB_init : BOOL
VAR_INPUT
	bInitRetains : BOOL; // if TRUE, the retain variables are initialized (warm start / cold start)
	bInCopyCode : BOOL;  // if TRUE, the instance afterwards gets moved into the copy code (online change)
END_VAR
AddInput('in1',THIS^.in1);
AddInput('in2',THIS^.in2);
AddOutput('out', THIS^.out);
END_METHOD

METHOD PROTECTED OnExecute
VAR
END_VAR
out.Value := LMOD(in1.Value, in2.Value);
END_METHOD

END_FUNCTION_BLOCK

// ---- Core/Nodes/MOD/MOD_LWORD.TcPOU
{attribute 'linkalways'} 
{attribute 'no_explicit_call' := 'This FB is a CLASS and must be accessed using methods or properties'}
{attribute 'enable_dynamic_creation'}
FUNCTION_BLOCK FINAL MOD_LWORD EXTENDS Node
VAR
	in1 : _LWORD(0);
	in2 : _LWORD(0);
	out : _LWORD(0);
END_VAR

METHOD PUBLIC Clone : I_Node
VAR
	pNode : POINTER TO MOD_LWORD;
END_VAR
pNode := __NEW(MOD_LWORD);
Clone := pNode^;
END_METHOD

METHOD FB_init : BOOL
VAR_INPUT
	bInitRetains : BOOL; // if TRUE, the retain variables are initialized (warm start / cold start)
	bInCopyCode : BOOL;  // if TRUE, the instance afterwards gets moved into the copy code (online change)
END_VAR
AddInput('in1',THIS^.in1);
AddInput('in2',THIS^.in2);
AddOutput('out', THIS^.out);
END_METHOD

METHOD PROTECTED OnExecute
VAR
END_VAR
out.Value := in1.Value MOD in2.Value;
END_METHOD

END_FUNCTION_BLOCK

// ---- Core/Nodes/MOD/MOD_SINT.TcPOU
{attribute 'linkalways'} 
{attribute 'no_explicit_call' := 'This FB is a CLASS and must be accessed using methods or properties'}
{attribute 'enable_dynamic_creation'}
FUNCTION_BLOCK FINAL MOD_SINT EXTENDS Node
VAR
	in1 : _SINT(0);
	in2 : _SINT(0);
	out : _SINT(0);
END_VAR

METHOD PUBLIC Clone : I_Node
VAR
	pNode : POINTER TO MOD_SINT;
END_VAR
pNode := __NEW(MOD_SINT);
Clone := pNode^;
END_METHOD

METHOD FB_init : BOOL
VAR_INPUT
	bInitRetains : BOOL; // if TRUE, the retain variables are initialized (warm start / cold start)
	bInCopyCode : BOOL;  // if TRUE, the instance afterwards gets moved into the copy code (online change)
END_VAR
AddInput('in1',THIS^.in1);
AddInput('in2',THIS^.in2);
AddOutput('out', THIS^.out);
END_METHOD

METHOD PROTECTED OnExecute
VAR
END_VAR
out.Value := in1.Value MOD in2.Value;
END_METHOD

END_FUNCTION_BLOCK

// ---- Core/Nodes/MOD/MOD_UDINT.TcPOU
{attribute 'linkalways'} 
{attribute 'no_explicit_call' := 'This FB is a CLASS and must be accessed using methods or properties'}
{attribute 'enable_dynamic_creation'}
FUNCTION_BLOCK FINAL MOD_UDINT EXTENDS Node
VAR
	in1 : _UDINT(0);
	in2 : _UDINT(0);
	out : _UDINT(0);
END_VAR

METHOD PUBLIC Clone : I_Node
VAR
	pNode : POINTER TO MOD_UDINT;
END_VAR
pNode := __NEW(MOD_UDINT);
Clone := pNode^;
END_METHOD

METHOD FB_init : BOOL
VAR_INPUT
	bInitRetains : BOOL; // if TRUE, the retain variables are initialized (warm start / cold start)
	bInCopyCode : BOOL;  // if TRUE, the instance afterwards gets moved into the copy code (online change)
END_VAR
AddInput('in1',THIS^.in1);
AddInput('in2',THIS^.in2);
AddOutput('out', THIS^.out);
END_METHOD

METHOD PROTECTED OnExecute
VAR
END_VAR
out.Value := in1.Value MOD in2.Value;
END_METHOD

END_FUNCTION_BLOCK

// ---- Core/Nodes/MOD/MOD_UINT.TcPOU
{attribute 'linkalways'} 
{attribute 'no_explicit_call' := 'This FB is a CLASS and must be accessed using methods or properties'}
{attribute 'enable_dynamic_creation'}
FUNCTION_BLOCK FINAL MOD_UINT EXTENDS Node
VAR
	in1 : _UINT(0);
	in2 : _UINT(0);
	out : _UINT(0);
END_VAR

METHOD PUBLIC Clone : I_Node
VAR
	pNode : POINTER TO MOD_UINT;
END_VAR
pNode := __NEW(MOD_UINT);
Clone := pNode^;
END_METHOD

METHOD FB_init : BOOL
VAR_INPUT
	bInitRetains : BOOL; // if TRUE, the retain variables are initialized (warm start / cold start)
	bInCopyCode : BOOL;  // if TRUE, the instance afterwards gets moved into the copy code (online change)
END_VAR
AddInput('in1',THIS^.in1);
AddInput('in2',THIS^.in2);
AddOutput('out', THIS^.out);
END_METHOD

METHOD PROTECTED OnExecute
VAR
END_VAR
out.Value := in1.Value MOD in2.Value;
END_METHOD

END_FUNCTION_BLOCK

// ---- Core/Nodes/MOD/MOD_ULINT.TcPOU
{attribute 'linkalways'} 
{attribute 'no_explicit_call' := 'This FB is a CLASS and must be accessed using methods or properties'}
{attribute 'enable_dynamic_creation'}
FUNCTION_BLOCK FINAL MOD_ULINT EXTENDS Node
VAR
	in1 : _ULINT(0);
	in2 : _ULINT(0);
	out : _ULINT(0);
END_VAR

METHOD PUBLIC Clone : I_Node
VAR
	pNode : POINTER TO MOD_ULINT;
END_VAR
pNode := __NEW(MOD_ULINT);
Clone := pNode^;
END_METHOD

METHOD FB_init : BOOL
VAR_INPUT
	bInitRetains : BOOL; // if TRUE, the retain variables are initialized (warm start / cold start)
	bInCopyCode : BOOL;  // if TRUE, the instance afterwards gets moved into the copy code (online change)
END_VAR
AddInput('in1',THIS^.in1);
AddInput('in2',THIS^.in2);
AddOutput('out', THIS^.out);
END_METHOD

METHOD PROTECTED OnExecute
VAR
END_VAR
out.Value := in1.Value MOD in2.Value;
END_METHOD

END_FUNCTION_BLOCK

// ---- Core/Nodes/MOD/MOD_USINT.TcPOU
{attribute 'linkalways'} 
{attribute 'no_explicit_call' := 'This FB is a CLASS and must be accessed using methods or properties'}
{attribute 'enable_dynamic_creation'}
FUNCTION_BLOCK FINAL MOD_USINT EXTENDS Node
VAR
	in1 : _USINT(0);
	in2 : _USINT(0);
	out : _USINT(0);
END_VAR

METHOD PUBLIC Clone : I_Node
VAR
	pNode : POINTER TO MOD_USINT;
END_VAR
pNode := __NEW(MOD_USINT);
Clone := pNode^;
END_METHOD

METHOD FB_init : BOOL
VAR_INPUT
	bInitRetains : BOOL; // if TRUE, the retain variables are initialized (warm start / cold start)
	bInCopyCode : BOOL;  // if TRUE, the instance afterwards gets moved into the copy code (online change)
END_VAR
AddInput('in1',THIS^.in1);
AddInput('in2',THIS^.in2);
AddOutput('out', THIS^.out);
END_METHOD

METHOD PROTECTED OnExecute
VAR
END_VAR
out.Value := in1.Value MOD in2.Value;
END_METHOD

END_FUNCTION_BLOCK

// ---- Core/Nodes/MOD/MOD_WORD.TcPOU
{attribute 'linkalways'} 
{attribute 'no_explicit_call' := 'This FB is a CLASS and must be accessed using methods or properties'}
{attribute 'enable_dynamic_creation'}
FUNCTION_BLOCK FINAL MOD_WORD EXTENDS Node
VAR
	in1 : _WORD(0);
	in2 : _WORD(0);
	out : _WORD(0);
END_VAR

METHOD PUBLIC Clone : I_Node
VAR
	pNode : POINTER TO MOD_WORD;
END_VAR
pNode := __NEW(MOD_WORD);
Clone := pNode^;
END_METHOD

METHOD FB_init : BOOL
VAR_INPUT
	bInitRetains : BOOL; // if TRUE, the retain variables are initialized (warm start / cold start)
	bInCopyCode : BOOL;  // if TRUE, the instance afterwards gets moved into the copy code (online change)
END_VAR
AddInput('in1',THIS^.in1);
AddInput('in2',THIS^.in2);
AddOutput('out', THIS^.out);
END_METHOD

METHOD PROTECTED OnExecute
VAR
END_VAR
out.Value := in1.Value MOD in2.Value;
END_METHOD

END_FUNCTION_BLOCK

// ---- Logic/MathLogicPack.TcPOU
{attribute 'linkalways'} 
{attribute 'no_explicit_call' := 'This FB is a CLASS and must be accessed using methods or properties'}
{attribute 'enable_dynamic_creation'}
FUNCTION_BLOCK MathLogicPack IMPLEMENTS I_GraphPack
VAR
	AND_BOOL : AND_BOOL;
	AND_BYTE : AND_BYTE;
	AND_DINT : AND_DINT;
	AND_DWORD : AND_DWORD;
	AND_INT : AND_INT;
	AND_LINT : AND_LINT;
	AND_LWORD : AND_LWORD;
	AND_SINT : AND_SINT;
	AND_UDINT : AND_UDINT;
	AND_UINT : AND_UINT;
	AND_ULINT : AND_ULINT;
	AND_USINT : AND_USINT;
	AND_WORD : AND_WORD;
	
	OR_BOOL : OR_BOOL;
	OR_BYTE : OR_BYTE;
	OR_DINT : OR_DINT;
	OR_DWORD : OR_DWORD;
	OR_INT : OR_INT;
	OR_LINT : OR_LINT;
	OR_LWORD : OR_LWORD;
	OR_SINT : OR_SINT;
	OR_UDINT : OR_UDINT;
	OR_UINT : OR_UINT;
	OR_ULINT : OR_ULINT;
	OR_USINT : OR_USINT;
	OR_WORD : OR_WORD;
	
	XOR_BOOL : XOR_BOOL;
	XOR_BYTE : XOR_BYTE;
	XOR_DINT : XOR_DINT;
	XOR_DWORD : XOR_DWORD;
	XOR_INT : XOR_INT;
	XOR_LINT : XOR_LINT;
	XOR_LWORD : XOR_LWORD;
	XOR_SINT : XOR_SINT;
	XOR_UDINT : XOR_UDINT;
	XOR_UINT : XOR_UINT;
	XOR_ULINT : XOR_ULINT;
	XOR_USINT : XOR_USINT;
	XOR_WORD : XOR_WORD;
	
	NOT_BOOL : NOT_BOOL;
	NOT_BYTE : NOT_BYTE;
	NOT_DINT : NOT_DINT;
	NOT_DWORD : NOT_DWORD;
	NOT_INT : NOT_INT;
	NOT_LINT : NOT_LINT;
	NOT_LWORD : NOT_LWORD;
	NOT_SINT : NOT_SINT;
	NOT_UDINT : NOT_UDINT;
	NOT_UINT : NOT_UINT;
	NOT_ULINT : NOT_ULINT;
	NOT_USINT : NOT_USINT;
	NOT_WORD : NOT_WORD;
END_VAR

METHOD Register
VAR_INPUT
	Datatypes : I_Datatypes;
	NodeFactory : I_NodeFactory;
END_VAR
NodeFactory.AddNodeAsPrototype('Math/Logic/AND/AND_BOOL',AND_BOOL);
NodeFactory.AddNodeAsPrototype('Math/Logic/AND/AND_BYTE',AND_BYTE);
NodeFactory.AddNodeAsPrototype('Math/Logic/AND/AND_DINT',AND_DINT);
NodeFactory.AddNodeAsPrototype('Math/Logic/AND/AND_DWORD',AND_DWORD);
NodeFactory.AddNodeAsPrototype('Math/Logic/AND/AND_INT',AND_INT);
NodeFactory.AddNodeAsPrototype('Math/Logic/AND/AND_LINT',AND_LINT);
NodeFactory.AddNodeAsPrototype('Math/Logic/AND/AND_LWORD',AND_LWORD);
NodeFactory.AddNodeAsPrototype('Math/Logic/AND/AND_SINT',AND_SINT);
NodeFactory.AddNodeAsPrototype('Math/Logic/AND/AND_UDINT',AND_UDINT);
NodeFactory.AddNodeAsPrototype('Math/Logic/AND/AND_UINT',AND_UINT);
NodeFactory.AddNodeAsPrototype('Math/Logic/AND/AND_ULINT',AND_ULINT);
NodeFactory.AddNodeAsPrototype('Math/Logic/AND/AND_USINT',AND_USINT);
NodeFactory.AddNodeAsPrototype('Math/Logic/AND/AND_WORD',AND_WORD);

NodeFactory.AddNodeAsPrototype('Math/Logic/OR/OR_BOOL',OR_BOOL);
NodeFactory.AddNodeAsPrototype('Math/Logic/OR/OR_BYTE',OR_BYTE);
NodeFactory.AddNodeAsPrototype('Math/Logic/OR/OR_DINT',OR_DINT);
NodeFactory.AddNodeAsPrototype('Math/Logic/OR/OR_DWORD',OR_DWORD);
NodeFactory.AddNodeAsPrototype('Math/Logic/OR/OR_INT',OR_INT);
NodeFactory.AddNodeAsPrototype('Math/Logic/OR/OR_LINT',OR_LINT);
NodeFactory.AddNodeAsPrototype('Math/Logic/OR/OR_LWORD',OR_LWORD);
NodeFactory.AddNodeAsPrototype('Math/Logic/OR/OR_SINT',OR_SINT);
NodeFactory.AddNodeAsPrototype('Math/Logic/OR/OR_UDINT',OR_UDINT);
NodeFactory.AddNodeAsPrototype('Math/Logic/OR/OR_UINT',OR_UINT);
NodeFactory.AddNodeAsPrototype('Math/Logic/OR/OR_ULINT',OR_ULINT);
NodeFactory.AddNodeAsPrototype('Math/Logic/OR/OR_USINT',OR_USINT);
NodeFactory.AddNodeAsPrototype('Math/Logic/OR/OR_WORD',OR_WORD);

NodeFactory.AddNodeAsPrototype('Math/Logic/XOR/XOR_BOOL',XOR_BOOL);
NodeFactory.AddNodeAsPrototype('Math/Logic/XOR/XOR_BYTE',XOR_BYTE);
NodeFactory.AddNodeAsPrototype('Math/Logic/XOR/XOR_DINT',XOR_DINT);
NodeFactory.AddNodeAsPrototype('Math/Logic/XOR/XOR_DWORD',XOR_DWORD);
NodeFactory.AddNodeAsPrototype('Math/Logic/XOR/XOR_INT',XOR_INT);
NodeFactory.AddNodeAsPrototype('Math/Logic/XOR/XOR_LINT',XOR_LINT);
NodeFactory.AddNodeAsPrototype('Math/Logic/XOR/XOR_LWORD',XOR_LWORD);
NodeFactory.AddNodeAsPrototype('Math/Logic/XOR/XOR_SINT',XOR_SINT);
NodeFactory.AddNodeAsPrototype('Math/Logic/XOR/XOR_UDINT',XOR_UDINT);
NodeFactory.AddNodeAsPrototype('Math/Logic/XOR/XOR_UINT',XOR_UINT);
NodeFactory.AddNodeAsPrototype('Math/Logic/XOR/XOR_ULINT',XOR_ULINT);
NodeFactory.AddNodeAsPrototype('Math/Logic/XOR/XOR_USINT',XOR_USINT);
NodeFactory.AddNodeAsPrototype('Math/Logic/XOR/XOR_WORD',XOR_WORD);

NodeFactory.AddNodeAsPrototype('Math/Logic/NOT/NOT_BOOL',NOT_BOOL);
NodeFactory.AddNodeAsPrototype('Math/Logic/NOT/NOT_BYTE',NOT_BYTE);
NodeFactory.AddNodeAsPrototype('Math/Logic/NOT/NOT_DINT',NOT_DINT);
NodeFactory.AddNodeAsPrototype('Math/Logic/NOT/NOT_DWORD',NOT_DWORD);
NodeFactory.AddNodeAsPrototype('Math/Logic/NOT/NOT_INT',NOT_INT);
NodeFactory.AddNodeAsPrototype('Math/Logic/NOT/NOT_LINT',NOT_LINT);
NodeFactory.AddNodeAsPrototype('Math/Logic/NOT/NOT_LWORD',NOT_LWORD);
NodeFactory.AddNodeAsPrototype('Math/Logic/NOT/NOT_SINT',NOT_SINT);
NodeFactory.AddNodeAsPrototype('Math/Logic/NOT/NOT_UDINT',NOT_UDINT);
NodeFactory.AddNodeAsPrototype('Math/Logic/NOT/NOT_UINT',NOT_UINT);
NodeFactory.AddNodeAsPrototype('Math/Logic/NOT/NOT_ULINT',NOT_ULINT);
NodeFactory.AddNodeAsPrototype('Math/Logic/NOT/NOT_USINT',NOT_USINT);
NodeFactory.AddNodeAsPrototype('Math/Logic/NOT/NOT_WORD',NOT_WORD);
END_METHOD

END_FUNCTION_BLOCK

// ---- Logic/Nodes/AND/AND_BOOL.TcPOU
{attribute 'linkalways'} 
{attribute 'no_explicit_call' := 'This FB is a CLASS and must be accessed using methods or properties'}
{attribute 'enable_dynamic_creation'}
FUNCTION_BLOCK FINAL AND_BOOL EXTENDS Node
VAR
	in1 : _BOOL(FALSE);
	in2 : _BOOL(FALSE);
	out : _BOOL(FALSE);
END_VAR

METHOD PUBLIC Clone : I_Node
VAR
	pNode : POINTER TO AND_BOOL;
END_VAR
pNode := __NEW(AND_BOOL);
Clone := pNode^;
END_METHOD

METHOD FB_init : BOOL
VAR_INPUT
	bInitRetains : BOOL; // if TRUE, the retain variables are initialized (warm start / cold start)
	bInCopyCode : BOOL;  // if TRUE, the instance afterwards gets moved into the copy code (online change)
END_VAR
AddInput('in1',THIS^.in1);
AddInput('in2',THIS^.in2);
AddOutput('out', THIS^.out);
END_METHOD

METHOD PROTECTED OnExecute
VAR
END_VAR
out.Value := in1.Value AND in2.Value;
END_METHOD

END_FUNCTION_BLOCK

// ---- Logic/Nodes/AND/AND_BYTE.TcPOU
{attribute 'linkalways'} 
{attribute 'no_explicit_call' := 'This FB is a CLASS and must be accessed using methods or properties'}
{attribute 'enable_dynamic_creation'}
FUNCTION_BLOCK FINAL AND_BYTE EXTENDS Node
VAR
	in1 : _BYTE(0);
	in2 : _BYTE(0);
	out : _BYTE(0);
END_VAR

METHOD PUBLIC Clone : I_Node
VAR
	pNode : POINTER TO AND_BYTE;
END_VAR
pNode := __NEW(AND_BYTE);
Clone := pNode^;
END_METHOD

METHOD FB_init : BOOL
VAR_INPUT
	bInitRetains : BOOL; // if TRUE, the retain variables are initialized (warm start / cold start)
	bInCopyCode : BOOL;  // if TRUE, the instance afterwards gets moved into the copy code (online change)
END_VAR
AddInput('in1',THIS^.in1);
AddInput('in2',THIS^.in2);
AddOutput('out', THIS^.out);
END_METHOD

METHOD PROTECTED OnExecute
VAR
END_VAR
out.Value := in1.Value AND in2.Value;
END_METHOD

END_FUNCTION_BLOCK

// ---- Logic/Nodes/AND/AND_DINT.TcPOU
{attribute 'linkalways'} 
{attribute 'no_explicit_call' := 'This FB is a CLASS and must be accessed using methods or properties'}
{attribute 'enable_dynamic_creation'}
FUNCTION_BLOCK FINAL AND_DINT EXTENDS Node
VAR
	in1 : _DINT(0);
	in2 : _DINT(0);
	out : _DINT(0);
END_VAR

METHOD PUBLIC Clone : I_Node
VAR
	pNode : POINTER TO AND_DINT;
END_VAR
pNode := __NEW(AND_DINT);
Clone := pNode^;
END_METHOD

METHOD FB_init : BOOL
VAR_INPUT
	bInitRetains : BOOL; // if TRUE, the retain variables are initialized (warm start / cold start)
	bInCopyCode : BOOL;  // if TRUE, the instance afterwards gets moved into the copy code (online change)
END_VAR
AddInput('in1',THIS^.in1);
AddInput('in2',THIS^.in2);
AddOutput('out', THIS^.out);
END_METHOD

METHOD PROTECTED OnExecute
VAR
END_VAR
out.Value := in1.Value AND in2.Value;
END_METHOD

END_FUNCTION_BLOCK

// ---- Logic/Nodes/AND/AND_DWORD.TcPOU
{attribute 'linkalways'} 
{attribute 'no_explicit_call' := 'This FB is a CLASS and must be accessed using methods or properties'}
{attribute 'enable_dynamic_creation'}
FUNCTION_BLOCK FINAL AND_DWORD EXTENDS Node
VAR
	in1 : _DWORD(0);
	in2 : _DWORD(0);
	out : _DWORD(0);
END_VAR

METHOD PUBLIC Clone : I_Node
VAR
	pNode : POINTER TO AND_DWORD;
END_VAR
pNode := __NEW(AND_DWORD);
Clone := pNode^;
END_METHOD

METHOD FB_init : BOOL
VAR_INPUT
	bInitRetains : BOOL; // if TRUE, the retain variables are initialized (warm start / cold start)
	bInCopyCode : BOOL;  // if TRUE, the instance afterwards gets moved into the copy code (online change)
END_VAR
AddInput('in1',THIS^.in1);
AddInput('in2',THIS^.in2);
AddOutput('out', THIS^.out);
END_METHOD

METHOD PROTECTED OnExecute
VAR
END_VAR
out.Value := in1.Value AND in2.Value;
END_METHOD

END_FUNCTION_BLOCK

// ---- Logic/Nodes/AND/AND_INT.TcPOU
{attribute 'linkalways'} 
{attribute 'no_explicit_call' := 'This FB is a CLASS and must be accessed using methods or properties'}
{attribute 'enable_dynamic_creation'}
FUNCTION_BLOCK FINAL AND_INT EXTENDS Node
VAR
	in1 : _INT(0);
	in2 : _INT(0);
	out : _INT(0);
END_VAR

METHOD PUBLIC Clone : I_Node
VAR
	pNode : POINTER TO AND_INT;
END_VAR
pNode := __NEW(AND_INT);
Clone := pNode^;
END_METHOD

METHOD FB_init : BOOL
VAR_INPUT
	bInitRetains : BOOL; // if TRUE, the retain variables are initialized (warm start / cold start)
	bInCopyCode : BOOL;  // if TRUE, the instance afterwards gets moved into the copy code (online change)
END_VAR
AddInput('in1',THIS^.in1);
AddInput('in2',THIS^.in2);
AddOutput('out', THIS^.out);
END_METHOD

METHOD PROTECTED OnExecute
VAR
END_VAR
out.Value := in1.Value AND in2.Value;
END_METHOD

END_FUNCTION_BLOCK

// ---- Logic/Nodes/AND/AND_LINT.TcPOU
{attribute 'linkalways'} 
{attribute 'no_explicit_call' := 'This FB is a CLASS and must be accessed using methods or properties'}
{attribute 'enable_dynamic_creation'}
FUNCTION_BLOCK FINAL AND_LINT EXTENDS Node
VAR
	in1 : _LINT(0);
	in2 : _LINT(0);
	out : _LINT(0);
END_VAR

METHOD PUBLIC Clone : I_Node
VAR
	pNode : POINTER TO AND_LINT;
END_VAR
pNode := __NEW(AND_LINT);
Clone := pNode^;
END_METHOD

METHOD FB_init : BOOL
VAR_INPUT
	bInitRetains : BOOL; // if TRUE, the retain variables are initialized (warm start / cold start)
	bInCopyCode : BOOL;  // if TRUE, the instance afterwards gets moved into the copy code (online change)
END_VAR
AddInput('in1',THIS^.in1);
AddInput('in2',THIS^.in2);
AddOutput('out', THIS^.out);
END_METHOD

METHOD PROTECTED OnExecute
VAR
END_VAR
out.Value := in1.Value AND in2.Value;
END_METHOD

END_FUNCTION_BLOCK

// ---- Logic/Nodes/AND/AND_LWORD.TcPOU
{attribute 'linkalways'} 
{attribute 'no_explicit_call' := 'This FB is a CLASS and must be accessed using methods or properties'}
{attribute 'enable_dynamic_creation'}
FUNCTION_BLOCK FINAL AND_LWORD EXTENDS Node
VAR
	in1 : _LWORD(0);
	in2 : _LWORD(0);
	out : _LWORD(0);
END_VAR

METHOD PUBLIC Clone : I_Node
VAR
	pNode : POINTER TO AND_LWORD;
END_VAR
pNode := __NEW(AND_LWORD);
Clone := pNode^;
END_METHOD

METHOD FB_init : BOOL
VAR_INPUT
	bInitRetains : BOOL; // if TRUE, the retain variables are initialized (warm start / cold start)
	bInCopyCode : BOOL;  // if TRUE, the instance afterwards gets moved into the copy code (online change)
END_VAR
AddInput('in1',THIS^.in1);
AddInput('in2',THIS^.in2);
AddOutput('out', THIS^.out);
END_METHOD

METHOD PROTECTED OnExecute
VAR
END_VAR
out.Value := in1.Value AND in2.Value;
END_METHOD

END_FUNCTION_BLOCK

// ---- Logic/Nodes/AND/AND_SINT.TcPOU
{attribute 'linkalways'} 
{attribute 'no_explicit_call' := 'This FB is a CLASS and must be accessed using methods or properties'}
{attribute 'enable_dynamic_creation'}
FUNCTION_BLOCK FINAL AND_SINT EXTENDS Node
VAR
	in1 : _SINT(0);
	in2 : _SINT(0);
	out : _SINT(0);
END_VAR

METHOD PUBLIC Clone : I_Node
VAR
	pNode : POINTER TO AND_SINT;
END_VAR
pNode := __NEW(AND_SINT);
Clone := pNode^;
END_METHOD

METHOD FB_init : BOOL
VAR_INPUT
	bInitRetains : BOOL; // if TRUE, the retain variables are initialized (warm start / cold start)
	bInCopyCode : BOOL;  // if TRUE, the instance afterwards gets moved into the copy code (online change)
END_VAR
AddInput('in1',THIS^.in1);
AddInput('in2',THIS^.in2);
AddOutput('out', THIS^.out);
END_METHOD

METHOD PROTECTED OnExecute
VAR
END_VAR
out.Value := in1.Value AND in2.Value;
END_METHOD

END_FUNCTION_BLOCK

// ---- Logic/Nodes/AND/AND_UDINT.TcPOU
{attribute 'linkalways'} 
{attribute 'no_explicit_call' := 'This FB is a CLASS and must be accessed using methods or properties'}
{attribute 'enable_dynamic_creation'}
FUNCTION_BLOCK FINAL AND_UDINT EXTENDS Node
VAR
	in1 : _UDINT(0);
	in2 : _UDINT(0);
	out : _UDINT(0);
END_VAR

METHOD PUBLIC Clone : I_Node
VAR
	pNode : POINTER TO AND_UDINT;
END_VAR
pNode := __NEW(AND_UDINT);
Clone := pNode^;
END_METHOD

METHOD FB_init : BOOL
VAR_INPUT
	bInitRetains : BOOL; // if TRUE, the retain variables are initialized (warm start / cold start)
	bInCopyCode : BOOL;  // if TRUE, the instance afterwards gets moved into the copy code (online change)
END_VAR
AddInput('in1',THIS^.in1);
AddInput('in2',THIS^.in2);
AddOutput('out', THIS^.out);
END_METHOD

METHOD PROTECTED OnExecute
VAR
END_VAR
out.Value := in1.Value AND in2.Value;
END_METHOD

END_FUNCTION_BLOCK

// ---- Logic/Nodes/AND/AND_UINT.TcPOU
{attribute 'linkalways'} 
{attribute 'no_explicit_call' := 'This FB is a CLASS and must be accessed using methods or properties'}
{attribute 'enable_dynamic_creation'}
FUNCTION_BLOCK FINAL AND_UINT EXTENDS Node
VAR
	in1 : _UINT(0);
	in2 : _UINT(0);
	out : _UINT(0);
END_VAR

METHOD PUBLIC Clone : I_Node
VAR
	pNode : POINTER TO AND_UINT;
END_VAR
pNode := __NEW(AND_UINT);
Clone := pNode^;
END_METHOD

METHOD FB_init : BOOL
VAR_INPUT
	bInitRetains : BOOL; // if TRUE, the retain variables are initialized (warm start / cold start)
	bInCopyCode : BOOL;  // if TRUE, the instance afterwards gets moved into the copy code (online change)
END_VAR
AddInput('in1',THIS^.in1);
AddInput('in2',THIS^.in2);
AddOutput('out', THIS^.out);
END_METHOD

METHOD PROTECTED OnExecute
VAR
END_VAR
out.Value := in1.Value AND in2.Value;
END_METHOD

END_FUNCTION_BLOCK

// ---- Logic/Nodes/AND/AND_ULINT.TcPOU
{attribute 'linkalways'} 
{attribute 'no_explicit_call' := 'This FB is a CLASS and must be accessed using methods or properties'}
{attribute 'enable_dynamic_creation'}
FUNCTION_BLOCK FINAL AND_ULINT EXTENDS Node
VAR
	in1 : _ULINT(0);
	in2 : _ULINT(0);
	out : _ULINT(0);
END_VAR

METHOD PUBLIC Clone : I_Node
VAR
	pNode : POINTER TO AND_ULINT;
END_VAR
pNode := __NEW(AND_ULINT);
Clone := pNode^;
END_METHOD

METHOD FB_init : BOOL
VAR_INPUT
	bInitRetains : BOOL; // if TRUE, the retain variables are initialized (warm start / cold start)
	bInCopyCode : BOOL;  // if TRUE, the instance afterwards gets moved into the copy code (online change)
END_VAR
AddInput('in1',THIS^.in1);
AddInput('in2',THIS^.in2);
AddOutput('out', THIS^.out);
END_METHOD

METHOD PROTECTED OnExecute
VAR
END_VAR
out.Value := in1.Value AND in2.Value;
END_METHOD

END_FUNCTION_BLOCK

// ---- Logic/Nodes/AND/AND_USINT.TcPOU
{attribute 'linkalways'} 
{attribute 'no_explicit_call' := 'This FB is a CLASS and must be accessed using methods or properties'}
{attribute 'enable_dynamic_creation'}
FUNCTION_BLOCK FINAL AND_USINT EXTENDS Node
VAR
	in1 : _USINT(0);
	in2 : _USINT(0);
	out : _USINT(0);
END_VAR

METHOD PUBLIC Clone : I_Node
VAR
	pNode : POINTER TO AND_USINT;
END_VAR
pNode := __NEW(AND_USINT);
Clone := pNode^;
END_METHOD

METHOD FB_init : BOOL
VAR_INPUT
	bInitRetains : BOOL; // if TRUE, the retain variables are initialized (warm start / cold start)
	bInCopyCode : BOOL;  // if TRUE, the instance afterwards gets moved into the copy code (online change)
END_VAR
AddInput('in1',THIS^.in1);
AddInput('in2',THIS^.in2);
AddOutput('out', THIS^.out);
END_METHOD

METHOD PROTECTED OnExecute
VAR
END_VAR
out.Value := in1.Value AND in2.Value;
END_METHOD

END_FUNCTION_BLOCK

// ---- Logic/Nodes/AND/AND_WORD.TcPOU
{attribute 'linkalways'} 
{attribute 'no_explicit_call' := 'This FB is a CLASS and must be accessed using methods or properties'}
{attribute 'enable_dynamic_creation'}
FUNCTION_BLOCK FINAL AND_WORD EXTENDS Node
VAR
	in1 : _WORD(0);
	in2 : _WORD(0);
	out : _WORD(0);
END_VAR

METHOD PUBLIC Clone : I_Node
VAR
	pNode : POINTER TO AND_WORD;
END_VAR
pNode := __NEW(AND_WORD);
Clone := pNode^;
END_METHOD

METHOD FB_init : BOOL
VAR_INPUT
	bInitRetains : BOOL; // if TRUE, the retain variables are initialized (warm start / cold start)
	bInCopyCode : BOOL;  // if TRUE, the instance afterwards gets moved into the copy code (online change)
END_VAR
AddInput('in1',THIS^.in1);
AddInput('in2',THIS^.in2);
AddOutput('out', THIS^.out);
END_METHOD

METHOD PROTECTED OnExecute
VAR
END_VAR
out.Value := in1.Value AND in2.Value;
END_METHOD

END_FUNCTION_BLOCK

// ---- Logic/Nodes/OR/OR_BOOL.TcPOU
{attribute 'linkalways'} 
{attribute 'no_explicit_call' := 'This FB is a CLASS and must be accessed using methods or properties'}
{attribute 'enable_dynamic_creation'}
FUNCTION_BLOCK FINAL OR_BOOL EXTENDS Node
VAR
	in1 : _BOOL(FALSE);
	in2 : _BOOL(FALSE);
	out : _BOOL(FALSE);
END_VAR

METHOD PUBLIC Clone : I_Node
VAR
	pNode : POINTER TO OR_BOOL;
END_VAR
pNode := __NEW(OR_BOOL);
Clone := pNode^;
END_METHOD

METHOD FB_init : BOOL
VAR_INPUT
	bInitRetains : BOOL; // if TRUE, the retain variables are initialized (warm start / cold start)
	bInCopyCode : BOOL;  // if TRUE, the instance afterwards gets moved into the copy code (online change)
END_VAR
AddInput('in1',THIS^.in1);
AddInput('in2',THIS^.in2);
AddOutput('out', THIS^.out);
END_METHOD

METHOD PROTECTED OnExecute
VAR
END_VAR
out.Value := in1.Value OR in2.Value;
END_METHOD

END_FUNCTION_BLOCK

// ---- Logic/Nodes/OR/OR_BYTE.TcPOU
{attribute 'linkalways'} 
{attribute 'no_explicit_call' := 'This FB is a CLASS and must be accessed using methods or properties'}
{attribute 'enable_dynamic_creation'}
FUNCTION_BLOCK FINAL OR_BYTE EXTENDS Node
VAR
	in1 : _BYTE(0);
	in2 : _BYTE(0);
	out : _BYTE(0);
END_VAR

METHOD PUBLIC Clone : I_Node
VAR
	pNode : POINTER TO OR_BYTE;
END_VAR
pNode := __NEW(OR_BYTE);
Clone := pNode^;
END_METHOD

METHOD FB_init : BOOL
VAR_INPUT
	bInitRetains : BOOL; // if TRUE, the retain variables are initialized (warm start / cold start)
	bInCopyCode : BOOL;  // if TRUE, the instance afterwards gets moved into the copy code (online change)
END_VAR
AddInput('in1',THIS^.in1);
AddInput('in2',THIS^.in2);
AddOutput('out', THIS^.out);
END_METHOD

METHOD PROTECTED OnExecute
VAR
END_VAR
out.Value := in1.Value OR in2.Value;
END_METHOD

END_FUNCTION_BLOCK

// ---- Logic/Nodes/OR/OR_DINT.TcPOU
{attribute 'linkalways'} 
{attribute 'no_explicit_call' := 'This FB is a CLASS and must be accessed using methods or properties'}
{attribute 'enable_dynamic_creation'}
FUNCTION_BLOCK FINAL OR_DINT EXTENDS Node
VAR
	in1 : _DINT(0);
	in2 : _DINT(0);
	out : _DINT(0);
END_VAR

METHOD PUBLIC Clone : I_Node
VAR
	pNode : POINTER TO OR_DINT;
END_VAR
pNode := __NEW(OR_DINT);
Clone := pNode^;
END_METHOD

METHOD FB_init : BOOL
VAR_INPUT
	bInitRetains : BOOL; // if TRUE, the retain variables are initialized (warm start / cold start)
	bInCopyCode : BOOL;  // if TRUE, the instance afterwards gets moved into the copy code (online change)
END_VAR
AddInput('in1',THIS^.in1);
AddInput('in2',THIS^.in2);
AddOutput('out', THIS^.out);
END_METHOD

METHOD PROTECTED OnExecute
VAR
END_VAR
out.Value := in1.Value OR in2.Value;
END_METHOD

END_FUNCTION_BLOCK

// ---- Logic/Nodes/OR/OR_DWORD.TcPOU
{attribute 'linkalways'} 
{attribute 'no_explicit_call' := 'This FB is a CLASS and must be accessed using methods or properties'}
{attribute 'enable_dynamic_creation'}
FUNCTION_BLOCK FINAL OR_DWORD EXTENDS Node
VAR
	in1 : _DWORD(0);
	in2 : _DWORD(0);
	out : _DWORD(0);
END_VAR

METHOD PUBLIC Clone : I_Node
VAR
	pNode : POINTER TO OR_DWORD;
END_VAR
pNode := __NEW(OR_DWORD);
Clone := pNode^;
END_METHOD

METHOD FB_init : BOOL
VAR_INPUT
	bInitRetains : BOOL; // if TRUE, the retain variables are initialized (warm start / cold start)
	bInCopyCode : BOOL;  // if TRUE, the instance afterwards gets moved into the copy code (online change)
END_VAR
AddInput('in1',THIS^.in1);
AddInput('in2',THIS^.in2);
AddOutput('out', THIS^.out);
END_METHOD

METHOD PROTECTED OnExecute
VAR
END_VAR
out.Value := in1.Value OR in2.Value;
END_METHOD

END_FUNCTION_BLOCK

// ---- Logic/Nodes/OR/OR_INT.TcPOU
{attribute 'linkalways'} 
{attribute 'no_explicit_call' := 'This FB is a CLASS and must be accessed using methods or properties'}
{attribute 'enable_dynamic_creation'}
FUNCTION_BLOCK FINAL OR_INT EXTENDS Node
VAR
	in1 : _INT(0);
	in2 : _INT(0);
	out : _INT(0);
END_VAR

METHOD PUBLIC Clone : I_Node
VAR
	pNode : POINTER TO OR_INT;
END_VAR
pNode := __NEW(OR_INT);
Clone := pNode^;
END_METHOD

METHOD FB_init : BOOL
VAR_INPUT
	bInitRetains : BOOL; // if TRUE, the retain variables are initialized (warm start / cold start)
	bInCopyCode : BOOL;  // if TRUE, the instance afterwards gets moved into the copy code (online change)
END_VAR
AddInput('in1',THIS^.in1);
AddInput('in2',THIS^.in2);
AddOutput('out', THIS^.out);
END_METHOD

METHOD PROTECTED OnExecute
VAR
END_VAR
out.Value := in1.Value OR in2.Value;
END_METHOD

END_FUNCTION_BLOCK

// ---- Logic/Nodes/OR/OR_LINT.TcPOU
{attribute 'linkalways'} 
{attribute 'no_explicit_call' := 'This FB is a CLASS and must be accessed using methods or properties'}
{attribute 'enable_dynamic_creation'}
FUNCTION_BLOCK FINAL OR_LINT EXTENDS Node
VAR
	in1 : _LINT(0);
	in2 : _LINT(0);
	out : _LINT(0);
END_VAR

METHOD PUBLIC Clone : I_Node
VAR
	pNode : POINTER TO OR_LINT;
END_VAR
pNode := __NEW(OR_LINT);
Clone := pNode^;
END_METHOD

METHOD FB_init : BOOL
VAR_INPUT
	bInitRetains : BOOL; // if TRUE, the retain variables are initialized (warm start / cold start)
	bInCopyCode : BOOL;  // if TRUE, the instance afterwards gets moved into the copy code (online change)
END_VAR
AddInput('in1',THIS^.in1);
AddInput('in2',THIS^.in2);
AddOutput('out', THIS^.out);
END_METHOD

METHOD PROTECTED OnExecute
VAR
END_VAR
out.Value := in1.Value OR in2.Value;
END_METHOD

END_FUNCTION_BLOCK

// ---- Logic/Nodes/OR/OR_LWORD.TcPOU
{attribute 'linkalways'} 
{attribute 'no_explicit_call' := 'This FB is a CLASS and must be accessed using methods or properties'}
{attribute 'enable_dynamic_creation'}
FUNCTION_BLOCK FINAL OR_LWORD EXTENDS Node
VAR
	in1 : _LWORD(0);
	in2 : _LWORD(0);
	out : _LWORD(0);
END_VAR

METHOD PUBLIC Clone : I_Node
VAR
	pNode : POINTER TO OR_LWORD;
END_VAR
pNode := __NEW(OR_LWORD);
Clone := pNode^;
END_METHOD

METHOD FB_init : BOOL
VAR_INPUT
	bInitRetains : BOOL; // if TRUE, the retain variables are initialized (warm start / cold start)
	bInCopyCode : BOOL;  // if TRUE, the instance afterwards gets moved into the copy code (online change)
END_VAR
AddInput('in1',THIS^.in1);
AddInput('in2',THIS^.in2);
AddOutput('out', THIS^.out);
END_METHOD

METHOD PROTECTED OnExecute
VAR
END_VAR
out.Value := in1.Value OR in2.Value;
END_METHOD

END_FUNCTION_BLOCK

// ---- Logic/Nodes/OR/OR_SINT.TcPOU
{attribute 'linkalways'} 
{attribute 'no_explicit_call' := 'This FB is a CLASS and must be accessed using methods or properties'}
{attribute 'enable_dynamic_creation'}
FUNCTION_BLOCK FINAL OR_SINT EXTENDS Node
VAR
	in1 : _SINT(0);
	in2 : _SINT(0);
	out : _SINT(0);
END_VAR

METHOD PUBLIC Clone : I_Node
VAR
	pNode : POINTER TO OR_SINT;
END_VAR
pNode := __NEW(OR_SINT);
Clone := pNode^;
END_METHOD

